Yaskawa INFORM job: A_ROOF_SIDE_0617_2_PAINT_33.JBI

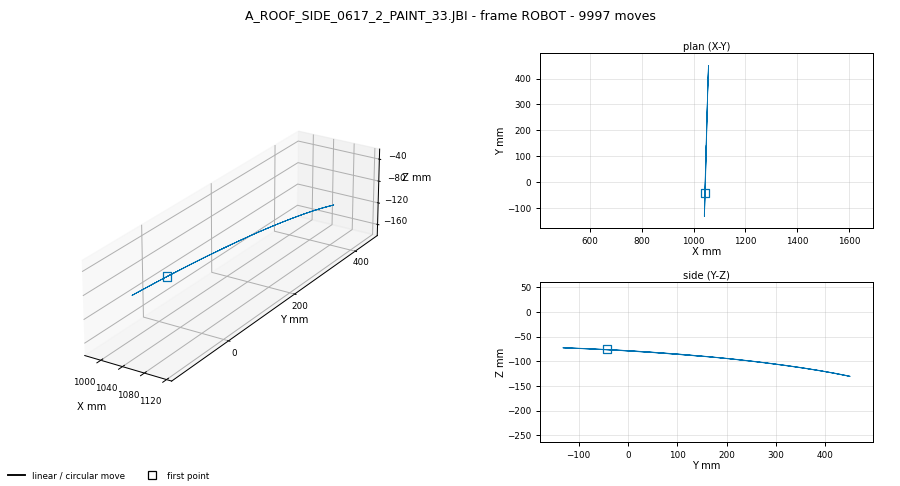
[picture p0: tool path of A_ROOF_SIDE_0617_2_PAINT_33.JBI in frame ROBOT, 9997 of 9997 moves have a stored position in this frame; points joined in program order, loops and branches not executed]
/JOB
//NAME A_ROOF_SIDE_0617_2_PAINT33
//POS
///NPOS 9997,0,0,0,0,0
///TOOL 1
///USER 0
///POSTYPE ROBOT
///RECTAN
///RCONF 1,0,0,0,0,0,0,0,0,0,0,0,0,0,0,0,0,0,0,0,0,0,0,0
C00000=1044.630,-42.557,-75.520,169.628,34.372,156.485
C00001=1044.636,-42.308,-75.534,169.630,34.372,156.485
C00002=1044.642,-42.058,-75.546,169.632,34.373,156.485
C00003=1044.648,-41.809,-75.559,169.634,34.375,156.485
C00004=1044.655,-41.560,-75.572,169.636,34.375,156.486
C00005=1044.661,-41.310,-75.585,169.638,34.376,156.486
C00006=1044.667,-41.061,-75.598,169.640,34.377,156.486
C00007=1044.674,-40.810,-75.611,169.642,34.378,156.486
C00008=1044.680,-40.561,-75.624,169.645,34.379,156.486
C00009=1044.687,-40.311,-75.636,169.647,34.380,156.486
C00010=1044.693,-40.062,-75.649,169.649,34.381,156.486
C00011=1044.699,-39.813,-75.663,169.651,34.382,156.486
C00012=1044.706,-39.562,-75.676,169.653,34.383,156.486
C00013=1044.712,-39.313,-75.689,169.656,34.384,156.487
C00014=1044.718,-39.063,-75.701,169.658,34.385,156.487
C00015=1044.725,-38.814,-75.714,169.660,34.385,156.487
C00016=1044.731,-38.565,-75.727,169.662,34.387,156.487
C00017=1044.738,-38.314,-75.740,169.664,34.388,156.487
C00018=1044.744,-38.065,-75.754,169.666,34.389,156.487
C00019=1044.749,-37.816,-75.767,169.668,34.390,156.487
C00020=1044.755,-37.566,-75.781,169.670,34.391,156.488
C00021=1044.761,-37.316,-75.793,169.672,34.392,156.488
C00022=1044.768,-37.067,-75.807,169.674,34.393,156.488
C00023=1044.774,-36.817,-75.820,169.677,34.394,156.488
C00024=1044.781,-36.568,-75.833,169.679,34.395,156.488
C00025=1044.787,-36.318,-75.846,169.681,34.396,156.488
C00026=1044.793,-36.069,-75.859,169.683,34.398,156.488
C00027=1044.800,-35.819,-75.873,169.685,34.398,156.489
C00028=1044.806,-35.538,-75.887,169.687,34.400,156.489
C00029=1044.813,-35.257,-75.903,169.689,34.401,156.489
C00030=1044.820,-34.977,-75.917,169.692,34.402,156.489
C00031=1044.828,-34.695,-75.932,169.694,34.403,156.489
C00032=1044.834,-34.446,-75.945,169.696,34.405,156.489
C00033=1044.840,-34.197,-75.958,169.698,34.405,156.489
C00034=1044.846,-33.947,-75.972,169.700,34.407,156.490
C00035=1044.852,-33.697,-75.986,169.702,34.407,156.490
C00036=1044.858,-33.448,-75.998,169.704,34.409,156.490
C00037=1044.864,-33.198,-76.012,169.706,34.410,156.490
C00038=1044.871,-32.949,-76.025,169.708,34.411,156.490
C00039=1044.878,-32.699,-76.039,169.710,34.412,156.490
C00040=1044.884,-32.450,-76.052,169.712,34.413,156.491
C00041=1044.890,-32.200,-76.065,169.714,34.414,156.491
C00042=1044.897,-31.951,-76.079,169.716,34.415,156.491
C00043=1044.903,-31.701,-76.092,169.718,34.416,156.491
C00044=1044.909,-31.452,-76.105,169.720,34.417,156.491
C00045=1044.915,-31.201,-76.119,169.722,34.418,156.491
C00046=1044.921,-30.952,-76.132,169.724,34.419,156.491
C00047=1044.927,-30.703,-76.145,169.726,34.420,156.491
C00048=1044.934,-30.453,-76.159,169.728,34.422,156.492
C00049=1044.940,-30.203,-76.172,169.730,34.422,156.492
C00050=1044.947,-29.954,-76.186,169.732,34.424,156.492
C00051=1044.953,-29.704,-76.199,169.734,34.424,156.492
C00052=1044.960,-29.455,-76.212,169.736,34.426,156.492
C00053=1044.966,-29.206,-76.226,169.739,34.427,156.492
C00054=1044.972,-28.955,-76.240,169.741,34.428,156.493
C00055=1044.978,-28.706,-76.253,169.743,34.429,156.493
C00056=1044.984,-28.457,-76.267,169.745,34.430,156.493
C00057=1044.991,-28.207,-76.280,169.748,34.431,156.493
C00058=1044.997,-27.958,-76.293,169.750,34.432,156.493
C00059=1045.004,-27.708,-76.307,169.752,34.434,156.493
C00060=1045.010,-27.458,-76.320,169.754,34.434,156.493
C00061=1045.017,-27.209,-76.334,169.756,34.436,156.494
C00062=1045.023,-26.959,-76.348,169.758,34.436,156.494
C00063=1045.029,-26.710,-76.361,169.760,34.438,156.494
C00064=1045.035,-26.461,-76.375,169.762,34.439,156.494
C00065=1045.042,-26.211,-76.389,169.763,34.440,156.494
C00066=1045.048,-25.961,-76.403,169.765,34.441,156.494
C00067=1045.054,-25.712,-76.416,169.767,34.443,156.495
C00068=1045.060,-25.462,-76.430,169.769,34.444,156.495
C00069=1045.066,-25.213,-76.443,169.771,34.445,156.495
C00070=1045.073,-24.963,-76.457,169.773,34.446,156.495
C00071=1045.079,-24.714,-76.472,169.775,34.447,156.495
C00072=1045.085,-24.464,-76.485,169.777,34.448,156.495
C00073=1045.091,-24.214,-76.499,169.779,34.450,156.496
C00074=1045.097,-23.965,-76.512,169.781,34.451,156.496
C00075=1045.104,-23.715,-76.526,169.783,34.452,156.496
C00076=1045.110,-23.465,-76.540,169.785,34.453,156.496
C00077=1045.116,-23.217,-76.554,169.787,34.454,156.496
C00078=1045.123,-22.967,-76.567,169.789,34.456,156.496
C00079=1045.128,-22.717,-76.581,169.791,34.457,156.497
C00080=1045.135,-22.467,-76.595,169.793,34.458,156.497
C00081=1045.141,-22.218,-76.610,169.795,34.459,156.497
C00082=1045.148,-21.968,-76.623,169.797,34.461,156.497
C00083=1045.154,-21.719,-76.636,169.799,34.461,156.497
C00084=1045.160,-21.469,-76.650,169.801,34.463,156.497
C00085=1045.167,-21.220,-76.665,169.804,34.464,156.498
C00086=1045.172,-20.970,-76.679,169.806,34.465,156.498
C00087=1045.179,-20.720,-76.692,169.808,34.466,156.498
C00088=1045.186,-20.472,-76.706,169.810,34.468,156.498
C00089=1045.192,-20.222,-76.720,169.812,34.469,156.498
C00090=1045.198,-19.972,-76.734,169.814,34.470,156.498
C00091=1045.204,-19.723,-76.749,169.816,34.471,156.499
C00092=1045.211,-19.441,-76.764,169.818,34.472,156.499
C00093=1045.218,-19.159,-76.780,169.820,34.474,156.499
C00094=1045.225,-18.878,-76.795,169.822,34.475,156.499
C00095=1045.232,-18.596,-76.811,169.824,34.477,156.499
C00096=1045.239,-18.347,-76.825,169.826,34.478,156.500
C00097=1045.245,-18.097,-76.839,169.828,34.479,156.500
C00098=1045.252,-17.848,-76.853,169.830,34.480,156.500
C00099=1045.258,-17.598,-76.867,169.832,34.481,156.500
C00100=1045.264,-17.348,-76.881,169.834,34.482,156.500
C00101=1045.271,-17.099,-76.895,169.836,34.484,156.500
C00102=1045.277,-16.849,-76.909,169.838,34.485,156.501
C00103=1045.284,-16.600,-76.923,169.840,34.486,156.501
C00104=1045.290,-16.350,-76.937,169.842,34.487,156.501
C00105=1045.296,-16.101,-76.951,169.844,34.488,156.501
C00106=1045.303,-15.851,-76.965,169.846,34.490,156.501
C00107=1045.308,-15.602,-76.979,169.848,34.491,156.502
C00108=1045.316,-15.352,-76.993,169.850,34.492,156.502
C00109=1045.322,-15.102,-77.007,169.852,34.493,156.502
C00110=1045.327,-14.853,-77.022,169.854,34.495,156.502
C00111=1045.334,-14.603,-77.036,169.855,34.496,156.502
C00112=1045.340,-14.354,-77.050,169.858,34.497,156.502
C00113=1045.346,-14.104,-77.064,169.860,34.499,156.503
C00114=1045.353,-13.855,-77.078,169.862,34.500,156.503
C00115=1045.359,-13.605,-77.093,169.864,34.501,156.503
C00116=1045.365,-13.356,-77.107,169.866,34.502,156.503
C00117=1045.372,-13.107,-77.122,169.868,34.503,156.503
C00118=1045.378,-12.856,-77.136,169.870,34.505,156.504
C00119=1045.383,-12.607,-77.150,169.872,34.506,156.504
C00120=1045.390,-12.357,-77.164,169.874,34.508,156.504
C00121=1045.396,-12.109,-77.179,169.876,34.509,156.504
C00122=1045.402,-11.859,-77.194,169.877,34.510,156.504
C00123=1045.409,-11.610,-77.207,169.879,34.512,156.505
C00124=1045.415,-11.360,-77.222,169.881,34.512,156.505
C00125=1045.421,-11.110,-77.236,169.883,34.514,156.505
C00126=1045.428,-10.861,-77.250,169.885,34.515,156.505
C00127=1045.434,-10.611,-77.265,169.887,34.516,156.505
C00128=1045.440,-10.361,-77.279,169.889,34.518,156.505
C00129=1045.447,-10.112,-77.293,169.891,34.519,156.506
C00130=1045.453,-9.863,-77.308,169.893,34.521,156.506
C00131=1045.459,-9.613,-77.322,169.895,34.522,156.506
C00132=1045.466,-9.364,-77.336,169.896,34.523,156.506
C00133=1045.472,-9.114,-77.351,169.898,34.525,156.507
C00134=1045.478,-8.865,-77.366,169.900,34.525,156.507
C00135=1045.484,-8.615,-77.380,169.903,34.527,156.507
C00136=1045.491,-8.366,-77.394,169.905,34.528,156.507
C00137=1045.497,-8.117,-77.409,169.907,34.529,156.507
C00138=1045.503,-7.866,-77.423,169.909,34.531,156.507
C00139=1045.510,-7.617,-77.438,169.911,34.532,156.508
C00140=1045.516,-7.368,-77.452,169.913,34.534,156.508
C00141=1045.522,-7.118,-77.467,169.914,34.535,156.508
C00142=1045.528,-6.868,-77.481,169.916,34.536,156.508
C00143=1045.535,-6.620,-77.495,169.918,34.537,156.508
C00144=1045.541,-6.370,-77.510,169.920,34.538,156.509
C00145=1045.548,-6.120,-77.525,169.922,34.540,156.509
C00146=1045.555,-5.871,-77.540,169.924,34.541,156.509
C00147=1045.560,-5.621,-77.553,169.926,34.542,156.509
C00148=1045.566,-5.372,-77.568,169.928,34.544,156.509
C00149=1045.573,-5.122,-77.583,169.929,34.545,156.510
C00150=1045.580,-4.873,-77.598,169.931,34.546,156.510
C00151=1045.586,-4.624,-77.612,169.933,34.548,156.510
C00152=1045.592,-4.373,-77.627,169.935,34.549,156.510
C00153=1045.598,-4.124,-77.641,169.937,34.551,156.510
C00154=1045.605,-3.875,-77.655,169.939,34.551,156.510
C00155=1045.611,-3.625,-77.670,169.941,34.553,156.511
C00156=1045.618,-3.342,-77.687,169.943,34.555,156.511
C00157=1045.626,-3.059,-77.704,169.946,34.556,156.511
C00158=1045.632,-2.775,-77.721,169.948,34.557,156.511
C00159=1045.639,-2.492,-77.738,169.950,34.559,156.512
C00160=1045.646,-2.243,-77.753,169.952,34.561,156.512
C00161=1045.651,-1.994,-77.767,169.954,34.562,156.512
C00162=1045.658,-1.744,-77.782,169.956,34.563,156.512
C00163=1045.664,-1.495,-77.797,169.957,34.565,156.513
C00164=1045.671,-1.245,-77.812,169.959,34.566,156.513
C00165=1045.676,-0.996,-77.827,169.961,34.567,156.513
C00166=1045.683,-0.746,-77.842,169.963,34.569,156.513
C00167=1045.689,-0.497,-77.857,169.965,34.570,156.513
C00168=1045.696,-0.247,-77.872,169.967,34.572,156.514
C00169=1045.701,0.002,-77.886,169.968,34.573,156.514
C00170=1045.708,0.252,-77.901,169.970,34.575,156.514
C00171=1045.713,0.502,-77.917,169.972,34.576,156.514
C00172=1045.720,0.751,-77.932,169.974,34.578,156.515
C00173=1045.726,1.000,-77.946,169.976,34.579,156.515
C00174=1045.732,1.250,-77.961,169.978,34.580,156.515
C00175=1045.738,1.500,-77.976,169.979,34.582,156.515
C00176=1045.745,1.749,-77.991,169.982,34.583,156.515
C00177=1045.750,1.998,-78.006,169.984,34.584,156.516
C00178=1045.757,2.248,-78.021,169.986,34.586,156.516
C00179=1045.763,2.497,-78.035,169.988,34.588,156.516
C00180=1045.770,2.746,-78.051,169.989,34.589,156.516
C00181=1045.776,2.996,-78.066,169.991,34.590,156.517
C00182=1045.783,3.246,-78.081,169.993,34.592,156.517
C00183=1045.788,3.495,-78.096,169.995,34.593,156.517
C00184=1045.795,3.744,-78.111,169.997,34.594,156.517
C00185=1045.801,3.994,-78.126,169.999,34.596,156.517
C00186=1045.807,4.244,-78.141,170.000,34.597,156.518
C00187=1045.814,4.493,-78.157,170.002,34.598,156.518
C00188=1045.820,4.743,-78.172,170.004,34.600,156.518
C00189=1045.826,4.992,-78.186,170.006,34.601,156.518
C00190=1045.832,5.241,-78.201,170.008,34.603,156.518
C00191=1045.839,5.491,-78.216,170.009,34.604,156.519
C00192=1045.845,5.740,-78.232,170.011,34.606,156.519
C00193=1045.852,5.990,-78.247,170.013,34.607,156.519
C00194=1045.858,6.239,-78.262,170.016,34.608,156.519
C00195=1045.864,6.489,-78.277,170.018,34.610,156.520
C00196=1045.869,6.738,-78.292,170.020,34.611,156.520
C00197=1045.876,6.987,-78.307,170.021,34.612,156.520
C00198=1045.882,7.237,-78.322,170.023,34.614,156.520
C00199=1045.889,7.487,-78.337,170.025,34.615,156.520
C00200=1045.895,7.736,-78.352,170.027,34.617,156.521
C00201=1045.902,7.985,-78.368,170.029,34.618,156.521
C00202=1045.908,8.235,-78.383,170.030,34.620,156.521
C00203=1045.915,8.485,-78.398,170.032,34.621,156.521
C00204=1045.921,8.734,-78.414,170.034,34.623,156.522
C00205=1045.927,8.984,-78.429,170.036,34.624,156.522
C00206=1045.933,9.233,-78.444,170.038,34.625,156.522
C00207=1045.940,9.482,-78.460,170.039,34.627,156.522
C00208=1045.946,9.731,-78.474,170.041,34.628,156.522
C00209=1045.952,9.981,-78.489,170.043,34.629,156.523
C00210=1045.959,10.230,-78.505,170.045,34.631,156.523
C00211=1045.965,10.480,-78.520,170.047,34.633,156.523
C00212=1045.971,10.730,-78.535,170.049,34.634,156.523
C00213=1045.978,10.979,-78.551,170.051,34.635,156.524
C00214=1045.984,11.228,-78.566,170.053,34.637,156.524
C00215=1045.990,11.478,-78.581,170.055,34.638,156.524
C00216=1045.997,11.727,-78.597,170.057,34.639,156.524
C00217=1046.004,11.977,-78.612,170.058,34.641,156.524
C00218=1046.010,12.226,-78.627,170.060,34.642,156.525
C00219=1046.016,12.476,-78.643,170.062,34.643,156.525
C00220=1046.023,12.761,-78.660,170.064,34.645,156.525
C00221=1046.031,13.046,-78.678,170.066,34.647,156.525
C00222=1046.038,13.331,-78.695,170.068,34.648,156.526
C00223=1046.045,13.616,-78.713,170.070,34.650,156.526
C00224=1046.052,13.865,-78.728,170.072,34.651,156.526
C00225=1046.058,14.115,-78.743,170.074,34.653,156.526
C00226=1046.065,14.364,-78.759,170.076,34.654,156.526
C00227=1046.070,14.614,-78.774,170.077,34.655,156.527
C00228=1046.077,14.863,-78.790,170.080,34.657,156.527
C00229=1046.083,15.113,-78.806,170.082,34.659,156.527
C00230=1046.090,15.362,-78.821,170.084,34.660,156.527
C00231=1046.096,15.611,-78.837,170.085,34.661,156.528
C00232=1046.102,15.861,-78.852,170.087,34.663,156.528
C00233=1046.109,16.110,-78.868,170.089,34.665,156.528
C00234=1046.114,16.360,-78.883,170.091,34.666,156.528
C00235=1046.121,16.609,-78.899,170.092,34.667,156.529
C00236=1046.127,16.859,-78.914,170.094,34.669,156.529
C00237=1046.133,17.108,-78.930,170.096,34.671,156.529
C00238=1046.140,17.357,-78.946,170.098,34.672,156.529
C00239=1046.146,17.607,-78.962,170.099,34.673,156.530
C00240=1046.152,17.856,-78.977,170.101,34.675,156.530
C00241=1046.159,18.107,-78.992,170.103,34.677,156.530
C00242=1046.165,18.356,-79.009,170.105,34.678,156.530
C00243=1046.172,18.605,-79.024,170.106,34.679,156.530
C00244=1046.177,18.855,-79.040,170.109,34.681,156.531
C00245=1046.184,19.104,-79.056,170.111,34.682,156.531
C00246=1046.191,19.353,-79.071,170.113,34.684,156.531
C00247=1046.197,19.603,-79.087,170.114,34.685,156.531
C00248=1046.203,19.852,-79.102,170.116,34.687,156.532
C00249=1046.209,20.101,-79.119,170.118,34.688,156.532
C00250=1046.216,20.351,-79.134,170.120,34.690,156.532
C00251=1046.221,20.600,-79.150,170.121,34.691,156.532
C00252=1046.228,20.849,-79.166,170.123,34.693,156.533
C00253=1046.234,21.099,-79.182,170.125,34.695,156.533
C00254=1046.240,21.349,-79.197,170.127,34.696,156.533
C00255=1046.246,21.598,-79.213,170.128,34.697,156.533
C00256=1046.253,21.848,-79.230,170.130,34.699,156.534
C00257=1046.260,22.097,-79.245,170.132,34.700,156.534
C00258=1046.265,22.347,-79.261,170.134,34.702,156.534
C00259=1046.272,22.596,-79.277,170.135,34.703,156.534
C00260=1046.278,22.845,-79.293,170.138,34.705,156.535
C00261=1046.285,23.094,-79.308,170.140,34.706,156.535
C00262=1046.291,23.344,-79.325,170.142,34.708,156.535
C00263=1046.296,23.594,-79.340,170.143,34.709,156.535
C00264=1046.303,23.843,-79.356,170.145,34.711,156.536
C00265=1046.310,24.093,-79.373,170.147,34.712,156.536
C00266=1046.316,24.342,-79.388,170.148,34.714,156.536
C00267=1046.322,24.591,-79.404,170.150,34.716,156.536
C00268=1046.329,24.841,-79.419,170.152,34.717,156.537
C00269=1046.334,25.090,-79.436,170.154,34.718,156.537
C00270=1046.340,25.339,-79.452,170.155,34.720,156.537
C00271=1046.347,25.588,-79.468,170.157,34.722,156.537
C00272=1046.354,25.839,-79.484,170.159,34.723,156.538
C00273=1046.360,26.088,-79.500,170.161,34.724,156.538
C00274=1046.366,26.337,-79.516,170.163,34.726,156.538
C00275=1046.373,26.586,-79.532,170.165,34.728,156.538
C00276=1046.379,26.835,-79.548,170.167,34.729,156.538
C00277=1046.385,27.085,-79.564,170.168,34.730,156.539
C00278=1046.392,27.335,-79.580,170.170,34.732,156.539
C00279=1046.398,27.584,-79.596,170.172,34.734,156.539
C00280=1046.404,27.834,-79.612,170.174,34.735,156.539
C00281=1046.410,28.083,-79.628,170.175,34.737,156.540
C00282=1046.416,28.332,-79.644,170.177,34.738,156.540
C00283=1046.423,28.582,-79.661,170.179,34.740,156.540
C00284=1046.430,28.868,-79.679,170.181,34.741,156.541
C00285=1046.438,29.155,-79.698,170.183,34.743,156.541
C00286=1046.445,29.440,-79.716,170.185,34.745,156.541
C00287=1046.451,29.727,-79.735,170.187,34.747,156.541
C00288=1046.458,29.977,-79.751,170.189,34.749,156.542
C00289=1046.464,30.226,-79.767,170.191,34.750,156.542
C00290=1046.470,30.476,-79.783,170.193,34.751,156.542
C00291=1046.476,30.725,-79.800,170.194,34.753,156.542
C00292=1046.482,30.974,-79.817,170.196,34.755,156.543
C00293=1046.490,31.224,-79.833,170.198,34.756,156.543
C00294=1046.496,31.473,-79.849,170.200,34.758,156.543
C00295=1046.502,31.722,-79.865,170.201,34.759,156.543
C00296=1046.507,31.972,-79.881,170.203,34.761,156.544
C00297=1046.514,32.222,-79.898,170.205,34.763,156.544
C00298=1046.521,32.471,-79.914,170.206,34.764,156.544
C00299=1046.527,32.720,-79.930,170.208,34.766,156.545
C00300=1046.533,32.969,-79.946,170.210,34.767,156.545
C00301=1046.539,33.219,-79.963,170.212,34.768,156.545
C00302=1046.545,33.468,-79.980,170.214,34.770,156.545
C00303=1046.552,33.717,-79.995,170.216,34.772,156.545
C00304=1046.558,33.967,-80.012,170.218,34.774,156.546
C00305=1046.565,34.217,-80.028,170.219,34.775,156.546
C00306=1046.571,34.466,-80.044,170.221,34.776,156.546
C00307=1046.577,34.715,-80.061,170.223,34.778,156.547
C00308=1046.583,34.964,-80.078,170.224,34.780,156.547
C00309=1046.590,35.214,-80.094,170.226,34.781,156.547
C00310=1046.596,35.463,-80.110,170.228,34.783,156.547
C00311=1046.602,35.713,-80.126,170.229,34.784,156.548
C00312=1046.609,35.963,-80.143,170.231,34.786,156.548
C00313=1046.615,36.211,-80.160,170.233,34.788,156.548
C00314=1046.621,36.461,-80.176,170.236,34.789,156.548
C00315=1046.628,36.710,-80.192,170.237,34.791,156.549
C00316=1046.634,36.960,-80.208,170.239,34.792,156.549
C00317=1046.640,37.208,-80.225,170.241,34.793,156.549
C00318=1046.646,37.458,-80.242,170.242,34.795,156.549
C00319=1046.653,37.708,-80.258,170.244,34.797,156.550
C00320=1046.659,37.957,-80.275,170.246,34.799,156.550
C00321=1046.665,38.206,-80.291,170.247,34.800,156.550
C00322=1046.671,38.456,-80.308,170.249,34.801,156.550
C00323=1046.677,38.705,-80.324,170.251,34.803,156.551
C00324=1046.684,38.954,-80.341,170.252,34.805,156.551
C00325=1046.690,39.204,-80.358,170.254,34.807,156.551
C00326=1046.697,39.453,-80.375,170.256,34.808,156.551
C00327=1046.702,39.702,-80.391,170.258,34.810,156.552
C00328=1046.709,39.952,-80.408,170.260,34.811,156.552
C00329=1046.715,40.201,-80.425,170.262,34.813,156.552
C00330=1046.720,40.451,-80.442,170.263,34.814,156.553
C00331=1046.727,40.701,-80.458,170.265,34.816,156.553
C00332=1046.733,40.949,-80.475,170.267,34.818,156.553
C00333=1046.739,41.199,-80.491,170.268,34.820,156.553
C00334=1046.746,41.448,-80.509,170.270,34.821,156.554
C00335=1046.752,41.698,-80.525,170.272,34.822,156.554
C00336=1046.758,41.947,-80.541,170.273,34.824,156.554
C00337=1046.765,42.196,-80.559,170.275,34.825,156.554
C00338=1046.771,42.446,-80.575,170.277,34.827,156.555
C00339=1046.777,42.694,-80.592,170.279,34.829,156.555
C00340=1046.784,42.944,-80.609,170.281,34.831,156.555
C00341=1046.790,43.193,-80.625,170.283,34.832,156.555
C00342=1046.796,43.443,-80.642,170.285,34.834,156.556
C00343=1046.802,43.692,-80.660,170.286,34.835,156.556
C00344=1046.808,43.942,-80.676,170.288,34.837,156.556
C00345=1046.815,44.191,-80.693,170.289,34.839,156.557
C00346=1046.820,44.441,-80.710,170.291,34.840,156.557
C00347=1046.826,44.689,-80.727,170.293,34.842,156.557
C00348=1046.833,44.977,-80.747,170.295,34.844,156.558
C00349=1046.840,45.263,-80.767,170.297,34.846,156.558
C00350=1046.848,45.549,-80.785,170.298,34.848,156.558
C00351=1046.855,45.835,-80.805,170.301,34.850,156.558
C00352=1046.861,46.085,-80.822,170.303,34.852,156.559
C00353=1046.867,46.334,-80.839,170.305,34.854,156.559
C00354=1046.873,46.583,-80.856,170.306,34.855,156.559
C00355=1046.879,46.833,-80.874,170.308,34.857,156.560
C00356=1046.885,47.082,-80.891,170.310,34.858,156.560
C00357=1046.891,47.331,-80.907,170.311,34.860,156.560
C00358=1046.897,47.581,-80.925,170.313,34.861,156.560
C00359=1046.904,47.830,-80.942,170.314,34.863,156.561
C00360=1046.910,48.080,-80.958,170.316,34.865,156.561
C00361=1046.916,48.329,-80.976,170.318,34.867,156.561
C00362=1046.922,48.578,-80.993,170.320,34.868,156.562
C00363=1046.928,48.827,-81.010,170.322,34.870,156.562
C00364=1046.934,49.076,-81.027,170.324,34.872,156.562
C00365=1046.941,49.326,-81.044,170.325,34.873,156.562
C00366=1046.947,49.575,-81.061,170.327,34.875,156.563
C00367=1046.953,49.825,-81.079,170.329,34.876,156.563
C00368=1046.959,50.074,-81.096,170.330,34.878,156.563
C00369=1046.966,50.324,-81.112,170.332,34.880,156.564
C00370=1046.971,50.573,-81.130,170.334,34.882,156.564
C00371=1046.978,50.822,-81.147,170.335,34.883,156.564
C00372=1046.984,51.071,-81.164,170.337,34.885,156.564
C00373=1046.990,51.321,-81.181,170.340,34.887,156.565
C00374=1046.996,51.570,-81.198,170.341,34.888,156.565
C00375=1047.003,51.819,-81.216,170.343,34.890,156.565
C00376=1047.009,52.068,-81.233,170.344,34.891,156.565
C00377=1047.015,52.318,-81.249,170.346,34.893,156.566
C00378=1047.021,52.568,-81.267,170.348,34.895,156.566
C00379=1047.028,52.817,-81.285,170.349,34.896,156.566
C00380=1047.034,53.066,-81.302,170.351,34.898,156.567
C00381=1047.040,53.315,-81.320,170.353,34.900,156.567
C00382=1047.046,53.565,-81.336,170.354,34.902,156.567
C00383=1047.053,53.814,-81.353,170.356,34.903,156.567
C00384=1047.058,54.063,-81.371,170.359,34.905,156.568
C00385=1047.065,54.313,-81.388,170.360,34.906,156.568
C00386=1047.071,54.562,-81.406,170.362,34.908,156.568
C00387=1047.078,54.811,-81.423,170.364,34.909,156.568
C00388=1047.084,55.060,-81.440,170.365,34.911,156.569
C00389=1047.090,55.310,-81.457,170.367,34.913,156.569
C00390=1047.096,55.559,-81.474,170.369,34.915,156.569
C00391=1047.103,55.808,-81.492,170.370,34.916,156.570
C00392=1047.109,56.058,-81.509,170.372,34.918,156.570
C00393=1047.115,56.307,-81.526,170.374,34.919,156.570
C00394=1047.121,56.557,-81.544,170.375,34.921,156.570
C00395=1047.128,56.805,-81.561,170.377,34.922,156.571
C00396=1047.134,57.055,-81.579,170.379,34.924,156.571
C00397=1047.140,57.304,-81.596,170.381,34.926,156.571
C00398=1047.147,57.553,-81.614,170.383,34.928,156.572
C00399=1047.153,57.804,-81.631,170.384,34.929,156.572
C00400=1047.159,58.052,-81.648,170.386,34.931,156.572
C00401=1047.166,58.302,-81.665,170.388,34.932,156.572
C00402=1047.171,58.551,-81.683,170.389,34.934,156.573
C00403=1047.178,58.800,-81.700,170.391,34.935,156.573
C00404=1047.184,59.050,-81.718,170.393,34.937,156.573
C00405=1047.190,59.299,-81.735,170.394,34.939,156.573
C00406=1047.197,59.548,-81.753,170.397,34.941,156.574
C00407=1047.203,59.798,-81.770,170.399,34.942,156.574
C00408=1047.210,60.047,-81.787,170.400,34.944,156.574
C00409=1047.216,60.296,-81.805,170.402,34.945,156.575
C00410=1047.223,60.546,-81.822,170.404,34.947,156.575
C00411=1047.228,60.795,-81.840,170.405,34.948,156.575
C00412=1047.236,61.081,-81.860,170.407,34.950,156.575
C00413=1047.244,61.366,-81.880,170.409,34.952,156.576
C00414=1047.251,61.652,-81.900,170.411,34.954,156.576
C00415=1047.258,61.939,-81.921,170.413,34.956,156.576
C00416=1047.264,62.188,-81.938,170.415,34.958,156.577
C00417=1047.271,62.438,-81.956,170.417,34.959,156.577
C00418=1047.278,62.687,-81.973,170.419,34.961,156.577
C00419=1047.283,62.936,-81.990,170.420,34.963,156.578
C00420=1047.290,63.185,-82.008,170.422,34.964,156.578
C00421=1047.296,63.435,-82.026,170.424,34.966,156.578
C00422=1047.303,63.684,-82.044,170.425,34.967,156.578
C00423=1047.309,63.933,-82.061,170.427,34.969,156.579
C00424=1047.316,64.182,-82.079,170.429,34.970,156.579
C00425=1047.322,64.432,-82.097,170.430,34.972,156.579
C00426=1047.327,64.681,-82.114,170.432,34.974,156.579
C00427=1047.334,64.931,-82.132,170.434,34.976,156.580
C00428=1047.341,65.180,-82.150,170.436,34.978,156.580
C00429=1047.346,65.429,-82.168,170.438,34.979,156.580
C00430=1047.352,65.679,-82.186,170.440,34.981,156.581
C00431=1047.359,65.928,-82.203,170.441,34.982,156.581
C00432=1047.365,66.177,-82.221,170.443,34.984,156.581
C00433=1047.371,66.426,-82.239,170.444,34.986,156.581
C00434=1047.378,66.676,-82.257,170.446,34.987,156.582
C00435=1047.384,66.925,-82.275,170.448,34.989,156.582
C00436=1047.389,67.174,-82.292,170.449,34.990,156.582
C00437=1047.396,67.423,-82.311,170.451,34.992,156.583
C00438=1047.403,67.673,-82.328,170.454,34.994,156.583
C00439=1047.408,67.922,-82.346,170.455,34.996,156.583
C00440=1047.415,68.171,-82.364,170.457,34.998,156.583
C00441=1047.421,68.421,-82.382,170.458,34.999,156.584
C00442=1047.428,68.670,-82.400,170.460,35.001,156.584
C00443=1047.433,68.919,-82.418,170.462,35.003,156.584
C00444=1047.440,69.168,-82.436,170.463,35.004,156.585
C00445=1047.446,69.418,-82.454,170.465,35.006,156.585
C00446=1047.453,69.667,-82.472,170.467,35.008,156.585
C00447=1047.458,69.916,-82.489,170.468,35.009,156.585
C00448=1047.465,70.166,-82.507,170.471,35.011,156.586
C00449=1047.471,70.415,-82.526,170.473,35.013,156.586
C00450=1047.476,70.664,-82.543,170.474,35.014,156.586
C00451=1047.483,70.913,-82.562,170.476,35.016,156.587
C00452=1047.489,71.163,-82.580,170.477,35.018,156.587
C00453=1047.495,71.413,-82.598,170.479,35.019,156.587
C00454=1047.502,71.661,-82.616,170.481,35.021,156.588
C00455=1047.508,71.910,-82.634,170.482,35.023,156.588
C00456=1047.514,72.159,-82.652,170.484,35.025,156.588
C00457=1047.520,72.409,-82.670,170.486,35.027,156.588
C00458=1047.526,72.658,-82.688,170.488,35.028,156.589
C00459=1047.532,72.907,-82.706,170.490,35.030,156.589
C00460=1047.539,73.157,-82.725,170.491,35.032,156.589
C00461=1047.545,73.406,-82.743,170.493,35.034,156.590
C00462=1047.551,73.655,-82.762,170.495,35.035,156.590
C00463=1047.557,73.904,-82.779,170.496,35.037,156.590
C00464=1047.563,74.154,-82.798,170.498,35.039,156.591
C00465=1047.569,74.403,-82.816,170.500,35.040,156.591
C00466=1047.576,74.652,-82.834,170.501,35.042,156.591
C00467=1047.583,74.902,-82.852,170.504,35.044,156.591
C00468=1047.588,75.150,-82.870,170.505,35.045,156.592
C00469=1047.595,75.400,-82.888,170.507,35.047,156.592
C00470=1047.601,75.649,-82.907,170.509,35.049,156.592
C00471=1047.607,75.899,-82.925,170.510,35.050,156.593
C00472=1047.614,76.148,-82.943,170.512,35.052,156.593
C00473=1047.620,76.398,-82.961,170.514,35.054,156.593
C00474=1047.626,76.646,-82.979,170.515,35.056,156.594
C00475=1047.632,76.895,-82.998,170.517,35.057,156.594
C00476=1047.639,77.182,-83.018,170.519,35.059,156.594
C00477=1047.646,77.468,-83.040,170.522,35.061,156.595
C00478=1047.653,77.753,-83.061,170.523,35.063,156.595
C00479=1047.660,78.039,-83.082,170.525,35.065,156.595
C00480=1047.667,78.288,-83.101,170.527,35.067,156.596
C00481=1047.673,78.538,-83.119,170.529,35.068,156.596
C00482=1047.679,78.786,-83.137,170.530,35.070,156.596
C00483=1047.684,79.036,-83.156,170.532,35.072,156.596
C00484=1047.691,79.286,-83.174,170.533,35.074,156.597
C00485=1047.697,79.535,-83.193,170.535,35.075,156.597
C00486=1047.703,79.784,-83.211,170.538,35.077,156.597
C00487=1047.710,80.033,-83.230,170.539,35.079,156.598
C00488=1047.715,80.282,-83.248,170.541,35.081,156.598
C00489=1047.721,80.531,-83.267,170.543,35.083,156.598
C00490=1047.728,80.781,-83.285,170.544,35.084,156.599
C00491=1047.734,81.030,-83.304,170.546,35.086,156.599
C00492=1047.740,81.279,-83.322,170.547,35.088,156.599
C00493=1047.746,81.529,-83.341,170.549,35.090,156.599
C00494=1047.752,81.778,-83.360,170.551,35.092,156.600
C00495=1047.759,82.027,-83.379,170.553,35.093,156.600
C00496=1047.764,82.276,-83.396,170.555,35.095,156.600
C00497=1047.771,82.525,-83.415,170.556,35.097,156.601
C00498=1047.777,82.774,-83.433,170.558,35.099,156.601
C00499=1047.783,83.024,-83.453,170.560,35.100,156.601
C00500=1047.789,83.273,-83.471,170.561,35.102,156.602
C00501=1047.796,83.522,-83.490,170.563,35.104,156.602
C00502=1047.802,83.772,-83.508,170.565,35.106,156.602
C00503=1047.807,84.021,-83.527,170.566,35.107,156.603
C00504=1047.814,84.270,-83.546,170.569,35.109,156.603
C00505=1047.820,84.519,-83.564,170.571,35.111,156.603
C00506=1047.826,84.768,-83.583,170.572,35.113,156.603
C00507=1047.832,85.017,-83.601,170.574,35.115,156.604
C00508=1047.838,85.266,-83.621,170.575,35.116,156.604
C00509=1047.845,85.516,-83.639,170.577,35.118,156.604
C00510=1047.851,85.765,-83.657,170.579,35.120,156.605
C00511=1047.857,86.014,-83.676,170.580,35.122,156.605
C00512=1047.863,86.264,-83.695,170.582,35.123,156.605
C00513=1047.869,86.513,-83.714,170.585,35.125,156.606
C00514=1047.876,86.762,-83.732,170.586,35.127,156.606
C00515=1047.882,87.011,-83.751,170.588,35.128,156.606
C00516=1047.888,87.261,-83.770,170.589,35.130,156.607
C00517=1047.894,87.510,-83.789,170.591,35.132,156.607
C00518=1047.901,87.759,-83.808,170.593,35.133,156.607
C00519=1047.907,88.008,-83.826,170.594,35.135,156.607
C00520=1047.913,88.257,-83.845,170.596,35.137,156.608
C00521=1047.919,88.507,-83.864,170.598,35.139,156.608
C00522=1047.926,88.756,-83.883,170.600,35.140,156.608
C00523=1047.932,89.005,-83.901,170.602,35.142,156.609
C00524=1047.938,89.254,-83.921,170.604,35.144,156.609
C00525=1047.944,89.503,-83.939,170.605,35.145,156.609
C00526=1047.951,89.753,-83.958,170.607,35.147,156.610
C00527=1047.957,90.002,-83.977,170.609,35.149,156.610
C00528=1047.963,90.251,-83.996,170.610,35.150,156.610
C00529=1047.969,90.500,-84.014,170.612,35.152,156.610
C00530=1047.975,90.750,-84.034,170.613,35.154,156.611
C00531=1047.981,90.999,-84.052,170.616,35.156,156.611
C00532=1047.987,91.248,-84.072,170.618,35.158,156.611
C00533=1047.993,91.497,-84.090,170.619,35.159,156.612
C00534=1047.999,91.747,-84.109,170.621,35.161,156.612
C00535=1048.006,91.995,-84.129,170.623,35.163,156.612
C00536=1048.011,92.245,-84.148,170.624,35.165,156.613
C00537=1048.018,92.494,-84.167,170.626,35.167,156.613
C00538=1048.024,92.743,-84.186,170.627,35.168,156.613
C00539=1048.030,92.992,-84.205,170.630,35.170,156.614
C00540=1048.037,93.278,-84.227,170.632,35.172,156.614
C00541=1048.045,93.564,-84.249,170.634,35.175,156.614
C00542=1048.051,93.849,-84.271,170.636,35.177,156.615
C00543=1048.058,94.136,-84.293,170.638,35.179,156.615
C00544=1048.064,94.385,-84.311,170.639,35.180,156.615
C00545=1048.070,94.634,-84.331,170.641,35.182,156.616
C00546=1048.077,94.883,-84.350,170.643,35.184,156.616
C00547=1048.082,95.133,-84.369,170.645,35.186,156.616
C00548=1048.089,95.382,-84.388,170.647,35.187,156.617
C00549=1048.095,95.630,-84.408,170.648,35.189,156.617
C00550=1048.101,95.880,-84.427,170.650,35.191,156.617
C00551=1048.107,96.129,-84.446,170.652,35.193,156.618
C00552=1048.114,96.379,-84.465,170.653,35.194,156.618
C00553=1048.120,96.628,-84.485,170.655,35.196,156.618
C00554=1048.126,96.877,-84.503,170.657,35.198,156.619
C00555=1048.132,97.126,-84.523,170.658,35.200,156.619
C00556=1048.138,97.376,-84.542,170.661,35.201,156.619
C00557=1048.144,97.624,-84.561,170.663,35.203,156.619
C00558=1048.150,97.874,-84.581,170.664,35.205,156.620
C00559=1048.156,98.123,-84.599,170.666,35.207,156.620
C00560=1048.162,98.371,-84.619,170.668,35.209,156.620
C00561=1048.170,98.621,-84.638,170.669,35.210,156.621
C00562=1048.175,98.871,-84.657,170.671,35.212,156.621
C00563=1048.182,99.119,-84.677,170.673,35.214,156.621
C00564=1048.188,99.369,-84.696,170.675,35.216,156.622
C00565=1048.194,99.617,-84.716,170.677,35.217,156.622
C00566=1048.200,99.867,-84.735,170.678,35.219,156.622
C00567=1048.206,100.116,-84.754,170.680,35.221,156.623
C00568=1048.213,100.365,-84.774,170.682,35.223,156.623
C00569=1048.219,100.615,-84.793,170.683,35.224,156.623
C00570=1048.224,100.864,-84.812,170.685,35.226,156.624
C00571=1048.230,101.113,-84.832,170.687,35.228,156.624
C00572=1048.237,101.362,-84.851,170.689,35.230,156.624
C00573=1048.243,101.611,-84.871,170.691,35.232,156.625
C00574=1048.249,101.860,-84.890,170.693,35.234,156.625
C00575=1048.255,102.110,-84.910,170.694,35.235,156.625
C00576=1048.261,102.359,-84.929,170.696,35.237,156.625
C00577=1048.268,102.608,-84.949,170.698,35.239,156.626
C00578=1048.273,102.857,-84.968,170.699,35.241,156.626
C00579=1048.279,103.106,-84.988,170.701,35.243,156.626
C00580=1048.285,103.355,-85.007,170.704,35.245,156.627
C00581=1048.291,103.604,-85.027,170.705,35.247,156.627
C00582=1048.298,103.854,-85.046,170.707,35.249,156.628
C00583=1048.304,104.103,-85.066,170.708,35.250,156.628
C00584=1048.310,104.352,-85.086,170.710,35.252,156.628
C00585=1048.316,104.601,-85.105,170.712,35.254,156.628
C00586=1048.322,104.850,-85.125,170.713,35.256,156.629
C00587=1048.327,105.099,-85.145,170.715,35.257,156.629
C00588=1048.335,105.349,-85.164,170.718,35.259,156.629
C00589=1048.340,105.598,-85.184,170.719,35.261,156.630
C00590=1048.346,105.847,-85.204,170.721,35.263,156.630
C00591=1048.352,106.096,-85.223,170.723,35.265,156.630
C00592=1048.358,106.345,-85.243,170.724,35.266,156.631
C00593=1048.365,106.595,-85.263,170.726,35.268,156.631
C00594=1048.371,106.843,-85.282,170.728,35.270,156.631
C00595=1048.377,107.093,-85.302,170.729,35.272,156.632
C00596=1048.383,107.341,-85.322,170.732,35.273,156.632
C00597=1048.390,107.591,-85.342,170.734,35.275,156.632
C00598=1048.395,107.840,-85.361,170.735,35.277,156.633
C00599=1048.401,108.089,-85.381,170.737,35.279,156.633
C00600=1048.407,108.338,-85.401,170.739,35.281,156.633
C00601=1048.414,108.588,-85.420,170.740,35.283,156.634
C00602=1048.420,108.837,-85.440,170.742,35.284,156.634
C00603=1048.426,109.085,-85.460,170.744,35.286,156.634
C00604=1048.433,109.371,-85.483,170.747,35.289,156.635
C00605=1048.440,109.657,-85.505,170.749,35.291,156.635
C00606=1048.447,109.943,-85.528,170.751,35.292,156.635
C00607=1048.455,110.229,-85.551,170.752,35.294,156.636
C00608=1048.461,110.478,-85.571,170.754,35.296,156.636
C00609=1048.467,110.728,-85.590,170.756,35.298,156.636
C00610=1048.473,110.977,-85.610,170.758,35.300,156.637
C00611=1048.479,111.225,-85.630,170.760,35.302,156.637
C00612=1048.485,111.475,-85.650,170.762,35.304,156.637
C00613=1048.491,111.724,-85.670,170.764,35.305,156.638
C00614=1048.497,111.973,-85.690,170.765,35.307,156.638
C00615=1048.503,112.222,-85.710,170.767,35.309,156.638
C00616=1048.510,112.471,-85.730,170.769,35.311,156.639
C00617=1048.516,112.720,-85.750,170.770,35.313,156.639
C00618=1048.522,112.969,-85.770,170.772,35.315,156.639
C00619=1048.528,113.219,-85.790,170.775,35.317,156.640
C00620=1048.534,113.467,-85.810,170.776,35.318,156.640
C00621=1048.540,113.717,-85.829,170.778,35.320,156.640
C00622=1048.547,113.966,-85.850,170.780,35.322,156.641
C00623=1048.553,114.215,-85.870,170.781,35.324,156.641
C00624=1048.558,114.464,-85.890,170.783,35.326,156.641
C00625=1048.564,114.713,-85.910,170.785,35.328,156.642
C00626=1048.570,114.963,-85.930,170.787,35.330,156.642
C00627=1048.576,115.212,-85.951,170.789,35.332,156.642
C00628=1048.582,115.461,-85.971,170.791,35.334,156.643
C00629=1048.588,115.710,-85.991,170.792,35.336,156.643
C00630=1048.594,115.959,-86.011,170.794,35.337,156.643
C00631=1048.599,116.208,-86.032,170.796,35.339,156.644
C00632=1048.605,116.457,-86.052,170.797,35.341,156.644
C00633=1048.612,116.706,-86.072,170.800,35.343,156.645
C00634=1048.618,116.955,-86.092,170.802,35.345,156.645
C00635=1048.623,117.204,-86.113,170.803,35.347,156.645
C00636=1048.630,117.454,-86.133,170.805,35.349,156.646
C00637=1048.636,117.703,-86.153,170.807,35.351,156.646
C00638=1048.641,117.952,-86.173,170.808,35.353,156.646
C00639=1048.648,118.201,-86.194,170.810,35.354,156.647
C00640=1048.654,118.450,-86.214,170.813,35.356,156.647
C00641=1048.660,118.698,-86.234,170.814,35.358,156.647
C00642=1048.666,118.948,-86.255,170.816,35.360,156.648
C00643=1048.672,119.197,-86.275,170.818,35.362,156.648
C00644=1048.679,119.446,-86.296,170.820,35.363,156.648
C00645=1048.684,119.696,-86.316,170.821,35.365,156.649
C00646=1048.690,119.944,-86.336,170.823,35.367,156.649
C00647=1048.696,120.194,-86.356,170.825,35.369,156.649
C00648=1048.702,120.443,-86.376,170.827,35.371,156.650
C00649=1048.708,120.692,-86.397,170.829,35.373,156.650
C00650=1048.715,120.941,-86.418,170.831,35.375,156.650
C00651=1048.721,121.189,-86.438,170.832,35.377,156.651
C00652=1048.726,121.439,-86.459,170.834,35.378,156.651
C00653=1048.732,121.688,-86.479,170.836,35.380,156.651
C00654=1048.738,121.937,-86.499,170.838,35.382,156.652
C00655=1048.745,122.186,-86.520,170.840,35.384,156.652
C00656=1048.751,122.435,-86.540,170.842,35.386,156.652
C00657=1048.757,122.684,-86.561,170.844,35.388,156.653
C00658=1048.762,122.934,-86.581,170.845,35.390,156.653
C00659=1048.769,123.183,-86.602,170.847,35.392,156.653
C00660=1048.775,123.431,-86.622,170.849,35.394,156.654
C00661=1048.781,123.681,-86.643,170.851,35.396,156.654
C00662=1048.787,123.930,-86.663,170.853,35.397,156.654
C00663=1048.793,124.179,-86.683,170.855,35.399,156.655
C00664=1048.799,124.428,-86.705,170.857,35.401,156.655
C00665=1048.805,124.677,-86.725,170.858,35.403,156.655
C00666=1048.812,124.926,-86.745,170.860,35.405,156.656
C00667=1048.817,125.175,-86.766,170.862,35.407,156.656
C00668=1048.825,125.462,-86.790,170.864,35.409,156.656
C00669=1048.832,125.747,-86.813,170.867,35.411,156.657
C00670=1048.839,126.032,-86.837,170.869,35.413,156.657
C00671=1048.846,126.318,-86.861,170.871,35.415,156.658
C00672=1048.852,126.567,-86.881,170.873,35.417,156.658
C00673=1048.858,126.816,-86.901,170.874,35.419,156.658
C00674=1048.864,127.065,-86.922,170.876,35.421,156.659
C00675=1048.870,127.314,-86.942,170.879,35.423,156.659
C00676=1048.876,127.564,-86.963,170.881,35.425,156.659
C00677=1048.883,127.812,-86.984,170.882,35.426,156.660
C00678=1048.889,128.062,-87.004,170.884,35.428,156.660
C00679=1048.895,128.310,-87.026,170.886,35.430,156.660
C00680=1048.901,128.560,-87.046,170.888,35.432,156.661
C00681=1048.908,128.809,-87.066,170.889,35.434,156.661
C00682=1048.914,129.058,-87.088,170.892,35.436,156.661
C00683=1048.920,129.307,-87.108,170.894,35.437,156.662
C00684=1048.926,129.555,-87.129,170.896,35.439,156.662
C00685=1048.932,129.805,-87.149,170.897,35.441,156.662
C00686=1048.938,130.054,-87.169,170.899,35.443,156.663
C00687=1048.944,130.303,-87.191,170.901,35.445,156.663
C00688=1048.951,130.553,-87.211,170.903,35.447,156.663
C00689=1048.957,130.801,-87.232,170.905,35.449,156.664
C00690=1048.963,131.051,-87.253,170.907,35.450,156.664
C00691=1048.970,131.299,-87.274,170.909,35.452,156.664
C00692=1048.975,131.549,-87.295,170.911,35.454,156.665
C00693=1048.982,131.798,-87.316,170.912,35.456,156.665
C00694=1048.988,132.047,-87.336,170.914,35.458,156.665
C00695=1048.994,132.296,-87.358,170.916,35.460,156.666
C00696=1049.000,132.544,-87.378,170.919,35.462,156.666
C00697=1049.006,132.794,-87.399,170.920,35.464,156.666
C00698=1049.011,133.042,-87.421,170.922,35.466,156.667
C00699=1049.018,133.292,-87.441,170.924,35.467,156.667
C00700=1049.024,133.541,-87.463,170.926,35.469,156.667
C00701=1049.030,133.790,-87.484,170.927,35.471,156.668
C00702=1049.036,134.039,-87.504,170.929,35.474,156.668
C00703=1049.042,134.288,-87.526,170.932,35.476,156.669
C00704=1049.048,134.537,-87.547,170.934,35.477,156.669
C00705=1049.054,134.786,-87.567,170.935,35.479,156.669
C00706=1049.060,135.035,-87.589,170.937,35.481,156.670
C00707=1049.066,135.284,-87.610,170.939,35.483,156.670
C00708=1049.072,135.533,-87.630,170.941,35.485,156.670
C00709=1049.079,135.782,-87.652,170.944,35.487,156.671
C00710=1049.085,136.031,-87.674,170.945,35.489,156.671
C00711=1049.091,136.280,-87.694,170.947,35.491,156.671
C00712=1049.097,136.529,-87.715,170.949,35.493,156.672
C00713=1049.102,136.778,-87.736,170.951,35.494,156.672
C00714=1049.109,137.027,-87.758,170.952,35.496,156.672
C00715=1049.115,137.277,-87.778,170.954,35.498,156.673
C00716=1049.121,137.525,-87.800,170.957,35.500,156.673
C00717=1049.127,137.774,-87.821,170.959,35.502,156.674
C00718=1049.133,138.024,-87.843,170.961,35.504,156.674
C00719=1049.139,138.272,-87.863,170.962,35.506,156.674
C00720=1049.145,138.522,-87.885,170.964,35.508,156.675
C00721=1049.151,138.771,-87.906,170.966,35.510,156.675
C00722=1049.157,139.019,-87.927,170.969,35.512,156.675
C00723=1049.164,139.268,-87.949,170.970,35.514,156.676
C00724=1049.170,139.518,-87.969,170.972,35.516,156.676
C00725=1049.175,139.766,-87.991,170.974,35.518,156.676
C00726=1049.181,140.016,-88.012,170.976,35.520,156.677
C00727=1049.188,140.265,-88.034,170.978,35.521,156.677
C00728=1049.193,140.513,-88.055,170.979,35.524,156.678
C00729=1049.199,140.763,-88.077,170.982,35.526,156.678
C00730=1049.205,141.012,-88.099,170.984,35.528,156.678
C00731=1049.212,141.260,-88.119,170.986,35.530,156.679
C00732=1049.219,141.546,-88.144,170.988,35.532,156.679
C00733=1049.225,141.831,-88.169,170.990,35.534,156.679
C00734=1049.232,142.117,-88.192,170.993,35.536,156.680
C00735=1049.239,142.403,-88.218,170.995,35.539,156.680
C00736=1049.246,142.652,-88.239,170.997,35.541,156.681
C00737=1049.251,142.900,-88.261,170.999,35.543,156.681
C00738=1049.257,143.150,-88.282,171.000,35.545,156.681
C00739=1049.263,143.399,-88.304,171.002,35.546,156.682
C00740=1049.269,143.647,-88.325,171.004,35.548,156.682
C00741=1049.275,143.896,-88.347,171.007,35.550,156.682
C00742=1049.281,144.146,-88.368,171.009,35.553,156.683
C00743=1049.287,144.395,-88.390,171.010,35.555,156.683
C00744=1049.293,144.643,-88.411,171.012,35.557,156.684
C00745=1049.299,144.893,-88.433,171.014,35.558,156.684
C00746=1049.305,145.142,-88.455,171.016,35.560,156.684
C00747=1049.312,145.391,-88.476,171.019,35.562,156.685
C00748=1049.318,145.639,-88.497,171.021,35.564,156.685
C00749=1049.324,145.888,-88.519,171.022,35.567,156.685
C00750=1049.330,146.138,-88.540,171.024,35.568,156.686
C00751=1049.336,146.387,-88.562,171.026,35.570,156.686
C00752=1049.343,146.635,-88.584,171.028,35.572,156.687
C00753=1049.348,146.884,-88.605,171.031,35.574,156.687
C00754=1049.355,147.133,-88.627,171.033,35.576,156.687
C00755=1049.361,147.382,-88.649,171.034,35.578,156.688
C00756=1049.367,147.632,-88.670,171.036,35.580,156.688
C00757=1049.373,147.881,-88.692,171.038,35.582,156.688
C00758=1049.378,148.130,-88.714,171.040,35.584,156.689
C00759=1049.384,148.378,-88.736,171.043,35.586,156.689
C00760=1049.390,148.627,-88.758,171.045,35.588,156.689
C00761=1049.397,148.877,-88.780,171.046,35.590,156.690
C00762=1049.403,149.126,-88.801,171.048,35.592,156.690
C00763=1049.408,149.374,-88.822,171.050,35.594,156.691
C00764=1049.415,149.623,-88.845,171.052,35.596,156.691
C00765=1049.421,149.872,-88.866,171.055,35.598,156.691
C00766=1049.426,150.122,-88.889,171.057,35.600,156.692
C00767=1049.433,150.371,-88.910,171.058,35.602,156.692
C00768=1049.438,150.619,-88.932,171.060,35.604,156.692
C00769=1049.445,150.868,-88.954,171.062,35.607,156.693
C00770=1049.451,151.117,-88.976,171.064,35.608,156.693
C00771=1049.456,151.366,-88.998,171.067,35.610,156.694
C00772=1049.463,151.615,-89.020,171.069,35.612,156.694
C00773=1049.469,151.864,-89.042,171.071,35.615,156.694
C00774=1049.475,152.113,-89.064,171.072,35.617,156.695
C00775=1049.481,152.361,-89.085,171.074,35.618,156.695
C00776=1049.486,152.611,-89.108,171.076,35.620,156.696
C00777=1049.493,152.860,-89.130,171.079,35.623,156.696
C00778=1049.499,153.109,-89.152,171.081,35.625,156.696
C00779=1049.505,153.358,-89.173,171.083,35.627,156.697
C00780=1049.511,153.607,-89.196,171.085,35.628,156.697
C00781=1049.517,153.856,-89.218,171.087,35.631,156.698
C00782=1049.523,154.105,-89.240,171.089,35.633,156.698
C00783=1049.529,154.353,-89.261,171.091,35.635,156.698
C00784=1049.534,154.603,-89.284,171.093,35.636,156.699
C00785=1049.541,154.851,-89.306,171.095,35.639,156.699
C00786=1049.547,155.100,-89.328,171.097,35.641,156.699
C00787=1049.554,155.349,-89.350,171.099,35.643,156.700
C00788=1049.559,155.599,-89.372,171.102,35.645,156.700
C00789=1049.565,155.847,-89.395,171.104,35.647,156.701
C00790=1049.571,156.097,-89.417,171.105,35.649,156.701
C00791=1049.577,156.345,-89.439,171.107,35.651,156.701
C00792=1049.583,156.594,-89.461,171.109,35.653,156.702
C00793=1049.589,156.843,-89.484,171.111,35.655,156.702
C00794=1049.595,157.092,-89.505,171.114,35.657,156.702
C00795=1049.601,157.340,-89.527,171.116,35.660,156.703
C00796=1049.608,157.626,-89.553,171.118,35.661,156.703
C00797=1049.615,157.911,-89.579,171.120,35.664,156.704
C00798=1049.622,158.197,-89.604,171.122,35.666,156.704
C00799=1049.629,158.481,-89.630,171.126,35.669,156.705
C00800=1049.635,158.730,-89.652,171.127,35.671,156.705
C00801=1049.641,158.979,-89.675,171.129,35.673,156.705
C00802=1049.647,159.229,-89.696,171.131,35.675,156.706
C00803=1049.653,159.477,-89.719,171.133,35.677,156.706
C00804=1049.659,159.726,-89.741,171.136,35.679,156.707
C00805=1049.665,159.975,-89.763,171.138,35.681,156.707
C00806=1049.672,160.224,-89.785,171.140,35.683,156.707
C00807=1049.677,160.473,-89.808,171.142,35.685,156.708
C00808=1049.683,160.722,-89.830,171.144,35.688,156.708
C00809=1049.689,160.971,-89.853,171.146,35.689,156.709
C00810=1049.695,161.220,-89.876,171.149,35.692,156.709
C00811=1049.701,161.469,-89.899,171.150,35.694,156.709
C00812=1049.706,161.718,-89.921,171.152,35.696,156.710
C00813=1049.712,161.967,-89.943,171.154,35.698,156.710
C00814=1049.718,162.216,-89.966,171.156,35.701,156.711
C00815=1049.724,162.465,-89.989,171.159,35.702,156.711
C00816=1049.729,162.714,-90.012,171.161,35.705,156.711
C00817=1049.736,162.963,-90.034,171.163,35.707,156.712
C00818=1049.742,163.212,-90.057,171.165,35.709,156.712
C00819=1049.747,163.460,-90.080,171.167,35.711,156.713
C00820=1049.753,163.709,-90.103,171.170,35.714,156.713
C00821=1049.759,163.957,-90.125,171.171,35.716,156.714
C00822=1049.765,164.206,-90.148,171.173,35.718,156.714
C00823=1049.770,164.456,-90.170,171.175,35.720,156.714
C00824=1049.776,164.705,-90.193,171.177,35.722,156.715
C00825=1049.782,164.953,-90.216,171.180,35.725,156.715
C00826=1049.788,165.202,-90.238,171.182,35.727,156.716
C00827=1049.794,165.451,-90.261,171.184,35.729,156.716
C00828=1049.799,165.700,-90.284,171.186,35.731,156.716
C00829=1049.806,165.949,-90.307,171.188,35.733,156.717
C00830=1049.812,166.198,-90.330,171.191,35.735,156.717
C00831=1049.818,166.447,-90.353,171.193,35.738,156.718
C00832=1049.824,166.696,-90.376,171.195,35.740,156.718
C00833=1049.829,166.945,-90.399,171.197,35.742,156.719
C00834=1049.835,167.194,-90.422,171.199,35.744,156.719
C00835=1049.841,167.442,-90.444,171.202,35.746,156.719
C00836=1049.847,167.691,-90.467,171.203,35.748,156.720
C00837=1049.853,167.940,-90.490,171.205,35.751,156.720
C00838=1049.859,168.189,-90.513,171.207,35.753,156.721
C00839=1049.865,168.438,-90.536,171.209,35.755,156.721
C00840=1049.870,168.687,-90.559,171.212,35.757,156.721
C00841=1049.877,168.935,-90.581,171.214,35.759,156.722
C00842=1049.882,169.184,-90.604,171.216,35.762,156.722
C00843=1049.888,169.433,-90.627,171.218,35.764,156.723
C00844=1049.895,169.683,-90.650,171.220,35.766,156.723
C00845=1049.900,169.932,-90.673,171.223,35.768,156.724
C00846=1049.906,170.180,-90.696,171.225,35.771,156.724
C00847=1049.912,170.429,-90.718,171.227,35.772,156.724
C00848=1049.918,170.678,-90.741,171.229,35.775,156.725
C00849=1049.924,170.926,-90.765,171.231,35.777,156.725
C00850=1049.930,171.175,-90.788,171.234,35.779,156.726
C00851=1049.936,171.425,-90.811,171.236,35.781,156.726
C00852=1049.942,171.674,-90.834,171.238,35.784,156.726
C00853=1049.949,171.922,-90.857,171.240,35.785,156.727
C00854=1049.954,172.171,-90.879,171.242,35.788,156.727
C00855=1049.960,172.419,-90.903,171.245,35.790,156.728
C00856=1049.966,172.668,-90.926,171.247,35.792,156.728
C00857=1049.972,172.918,-90.949,171.249,35.795,156.729
C00858=1049.978,173.167,-90.972,171.251,35.797,156.729
C00859=1049.984,173.416,-90.995,171.253,35.799,156.729
C00860=1049.991,173.699,-91.022,171.256,35.802,156.730
C00861=1049.998,173.985,-91.048,171.259,35.804,156.730
C00862=1050.005,174.269,-91.075,171.261,35.807,156.731
C00863=1050.012,174.554,-91.101,171.263,35.809,156.731
C00864=1050.017,174.803,-91.124,171.265,35.811,156.732
C00865=1050.024,175.052,-91.147,171.268,35.813,156.732
C00866=1050.031,175.301,-91.171,171.270,35.816,156.733
C00867=1050.036,175.550,-91.194,171.272,35.818,156.733
C00868=1050.042,175.798,-91.217,171.274,35.820,156.733
C00869=1050.048,176.047,-91.240,171.277,35.822,156.734
C00870=1050.054,176.296,-91.264,171.280,35.824,156.734
C00871=1050.060,176.545,-91.287,171.282,35.826,156.735
C00872=1050.066,176.794,-91.310,171.284,35.829,156.735
C00873=1050.072,177.042,-91.333,171.286,35.831,156.735
C00874=1050.079,177.292,-91.356,171.289,35.833,156.736
C00875=1050.085,177.540,-91.380,171.291,35.836,156.736
C00876=1050.091,177.789,-91.402,171.293,35.837,156.737
C00877=1050.097,178.038,-91.426,171.295,35.840,156.737
C00878=1050.103,178.287,-91.449,171.297,35.842,156.738
C00879=1050.109,178.536,-91.472,171.300,35.844,156.738
C00880=1050.115,178.785,-91.496,171.302,35.846,156.738
C00881=1050.121,179.034,-91.519,171.304,35.849,156.739
C00882=1050.127,179.282,-91.543,171.306,35.850,156.739
C00883=1050.134,179.531,-91.566,171.308,35.853,156.740
C00884=1050.140,179.779,-91.589,171.311,35.855,156.740
C00885=1050.146,180.028,-91.612,171.313,35.857,156.741
C00886=1050.153,180.277,-91.636,171.316,35.860,156.741
C00887=1050.158,180.526,-91.659,171.318,35.861,156.741
C00888=1050.165,180.775,-91.683,171.320,35.864,156.742
C00889=1050.171,181.024,-91.706,171.323,35.866,156.742
C00890=1050.177,181.272,-91.730,171.325,35.868,156.743
C00891=1050.183,181.522,-91.753,171.327,35.871,156.743
C00892=1050.189,181.770,-91.777,171.329,35.873,156.744
C00893=1050.196,182.020,-91.800,171.332,35.875,156.744
C00894=1050.202,182.268,-91.824,171.334,35.877,156.744
C00895=1050.208,182.516,-91.848,171.336,35.879,156.745
C00896=1050.214,182.766,-91.871,171.339,35.882,156.745
C00897=1050.220,183.014,-91.895,171.341,35.884,156.746
C00898=1050.226,183.264,-91.918,171.344,35.886,156.746
C00899=1050.233,183.512,-91.941,171.346,35.888,156.747
C00900=1050.240,183.761,-91.965,171.348,35.890,156.747
C00901=1050.245,184.010,-91.988,171.350,35.893,156.748
C00902=1050.251,184.258,-92.012,171.352,35.895,156.748
C00903=1050.257,184.507,-92.036,171.355,35.897,156.748
C00904=1050.262,184.756,-92.060,171.357,35.900,156.749
C00905=1050.268,185.005,-92.083,171.359,35.902,156.749
C00906=1050.274,185.254,-92.108,171.361,35.905,156.750
C00907=1050.280,185.502,-92.132,171.365,35.907,156.750
C00908=1050.286,185.751,-92.156,171.367,35.909,156.751
C00909=1050.292,186.000,-92.179,171.369,35.912,156.751
C00910=1050.298,186.249,-92.203,171.371,35.914,156.752
C00911=1050.304,186.498,-92.227,171.374,35.916,156.752
C00912=1050.310,186.746,-92.251,171.376,35.919,156.753
C00913=1050.315,186.995,-92.275,171.378,35.921,156.753
C00914=1050.322,187.244,-92.299,171.380,35.924,156.753
C00915=1050.327,187.492,-92.324,171.383,35.926,156.754
C00916=1050.333,187.741,-92.347,171.385,35.929,156.754
C00917=1050.339,187.991,-92.371,171.388,35.931,156.755
C00918=1050.345,188.239,-92.395,171.390,35.933,156.755
C00919=1050.351,188.488,-92.420,171.392,35.936,156.756
C00920=1050.357,188.736,-92.443,171.395,35.938,156.756
C00921=1050.363,188.986,-92.468,171.397,35.941,156.757
C00922=1050.369,189.234,-92.491,171.399,35.943,156.757
C00923=1050.374,189.483,-92.516,171.401,35.945,156.758
C00924=1050.381,189.767,-92.543,171.405,35.948,156.758
C00925=1050.388,190.052,-92.571,171.407,35.951,156.759
C00926=1050.395,190.336,-92.598,171.410,35.954,156.759
C00927=1050.402,190.620,-92.626,171.413,35.956,156.760
C00928=1050.408,190.869,-92.650,171.415,35.959,156.760
C00929=1050.414,191.118,-92.675,171.417,35.961,156.761
C00930=1050.419,191.366,-92.699,171.420,35.963,156.761
C00931=1050.426,191.615,-92.723,171.422,35.966,156.762
C00932=1050.431,191.864,-92.747,171.425,35.968,156.762
C00933=1050.438,192.113,-92.771,171.427,35.971,156.763
C00934=1050.443,192.361,-92.795,171.429,35.973,156.763
C00935=1050.450,192.610,-92.819,171.431,35.976,156.764
C00936=1050.455,192.859,-92.844,171.435,35.978,156.764
C00937=1050.462,193.108,-92.868,171.437,35.981,156.765
C00938=1050.467,193.356,-92.892,171.439,35.983,156.765
C00939=1050.474,193.605,-92.917,171.441,35.986,156.766
C00940=1050.479,193.853,-92.941,171.444,35.988,156.766
C00941=1050.485,194.103,-92.966,171.446,35.990,156.767
C00942=1050.492,194.352,-92.990,171.449,35.993,156.767
C00943=1050.497,194.600,-93.014,171.451,35.995,156.768
C00944=1050.504,194.849,-93.038,171.454,35.998,156.768
C00945=1050.510,195.097,-93.063,171.456,36.000,156.769
C00946=1050.516,195.346,-93.087,171.458,36.002,156.769
C00947=1050.522,195.595,-93.111,171.461,36.005,156.769
C00948=1050.528,195.844,-93.135,171.464,36.007,156.770
C00949=1050.534,196.092,-93.160,171.466,36.009,156.770
C00950=1050.540,196.341,-93.184,171.468,36.012,156.771
C00951=1050.546,196.590,-93.209,171.470,36.014,156.771
C00952=1050.552,196.839,-93.233,171.474,36.017,156.772
C00953=1050.558,197.087,-93.258,171.476,36.019,156.772
C00954=1050.564,197.336,-93.282,171.478,36.022,156.773
C00955=1050.571,197.585,-93.306,171.480,36.024,156.773
C00956=1050.577,197.833,-93.331,171.484,36.027,156.774
C00957=1050.583,198.082,-93.355,171.486,36.029,156.774
C00958=1050.589,198.331,-93.380,171.488,36.031,156.775
C00959=1050.595,198.579,-93.405,171.490,36.034,156.775
C00960=1050.601,198.828,-93.429,171.494,36.036,156.776
C00961=1050.607,199.078,-93.454,171.496,36.039,156.776
C00962=1050.614,199.325,-93.478,171.498,36.042,156.777
C00963=1050.620,199.575,-93.503,171.500,36.044,156.777
C00964=1050.625,199.824,-93.527,171.504,36.047,156.778
C00965=1050.632,200.072,-93.552,171.506,36.049,156.778
C00966=1050.638,200.321,-93.576,171.508,36.052,156.779
C00967=1050.645,200.569,-93.601,171.510,36.054,156.779
C00968=1050.651,200.818,-93.626,171.514,36.056,156.780
C00969=1050.657,201.067,-93.651,171.516,36.059,156.780
C00970=1050.663,201.315,-93.675,171.518,36.061,156.781
C00971=1050.669,201.564,-93.700,171.520,36.064,156.781
C00972=1050.675,201.813,-93.725,171.524,36.066,156.782
C00973=1050.681,202.062,-93.750,171.526,36.069,156.782
C00974=1050.687,202.310,-93.774,171.528,36.072,156.783
C00975=1050.693,202.559,-93.799,171.531,36.074,156.783
C00976=1050.699,202.808,-93.824,171.534,36.077,156.784
C00977=1050.705,203.056,-93.849,171.536,36.079,156.784
C00978=1050.711,203.305,-93.874,171.538,36.081,156.785
C00979=1050.717,203.554,-93.898,171.541,36.084,156.785
C00980=1050.723,203.803,-93.924,171.544,36.087,156.786
C00981=1050.729,204.051,-93.949,171.546,36.089,156.786
C00982=1050.735,204.300,-93.973,171.548,36.092,156.787
C00983=1050.741,204.549,-93.999,171.552,36.095,156.787
C00984=1050.747,204.797,-94.024,171.554,36.097,156.788
C00985=1050.752,205.046,-94.048,171.556,36.100,156.788
C00986=1050.759,205.294,-94.073,171.559,36.103,156.789
C00987=1050.766,205.543,-94.098,171.562,36.105,156.789
C00988=1050.790,206.596,-94.204,171.789,36.201,156.808
C00989=1050.797,206.846,-94.231,171.790,36.205,156.809
C00990=1050.804,207.098,-94.257,171.793,36.208,156.809
C00991=1050.810,207.349,-94.283,171.795,36.211,156.810
C00992=1050.817,207.600,-94.309,171.797,36.215,156.811
C00993=1050.824,207.849,-94.336,171.799,36.218,156.812
C00994=1050.829,208.098,-94.362,171.801,36.221,156.812
C00995=1050.836,208.346,-94.388,171.803,36.225,156.813
C00996=1050.843,208.594,-94.414,171.805,36.228,156.814
C00997=1050.849,208.843,-94.441,171.806,36.232,156.814
C00998=1050.855,209.092,-94.466,171.809,36.235,156.815
C00999=1050.862,209.340,-94.493,171.811,36.238,156.816
C01000=1050.869,209.588,-94.519,171.813,36.242,156.816
C01001=1050.874,209.837,-94.545,171.815,36.245,156.817
C01002=1050.881,210.086,-94.571,171.816,36.248,156.818
C01003=1050.888,210.334,-94.597,171.819,36.252,156.819
C01004=1050.893,210.582,-94.624,171.821,36.256,156.819
C01005=1050.901,210.831,-94.650,171.823,36.259,156.820
C01006=1050.906,211.080,-94.676,171.825,36.262,156.821
C01007=1050.913,211.329,-94.702,171.827,36.266,156.821
C01008=1050.920,211.577,-94.728,171.829,36.269,156.822
C01009=1050.925,211.825,-94.755,171.831,36.272,156.823
C01010=1050.933,212.074,-94.782,171.832,36.275,156.823
C01011=1050.938,212.322,-94.808,171.835,36.279,156.824
C01012=1050.945,212.570,-94.834,171.837,36.283,156.825
C01013=1050.951,212.820,-94.861,171.839,36.286,156.825
C01014=1050.957,213.068,-94.887,171.841,36.289,156.826
C01015=1050.964,213.317,-94.914,171.843,36.293,156.827
C01016=1050.970,213.565,-94.940,171.845,36.296,156.828
C01017=1050.976,213.814,-94.966,171.847,36.299,156.828
C01018=1050.983,214.062,-94.993,171.850,36.303,156.829
C01019=1050.989,214.311,-95.019,171.851,36.306,156.830
C01020=1050.996,214.560,-95.046,171.853,36.310,156.830
C01021=1051.002,214.808,-95.072,171.856,36.313,156.831
C01022=1051.008,215.056,-95.099,171.857,36.316,156.832
C01023=1051.015,215.305,-95.126,171.860,36.320,156.832
C01024=1051.021,215.553,-95.152,171.862,36.323,156.833
C01025=1051.028,215.802,-95.179,171.863,36.326,156.834
C01026=1051.033,216.050,-95.205,171.866,36.330,156.835
C01027=1051.041,216.299,-95.232,171.868,36.333,156.835
C01028=1051.046,216.548,-95.258,171.870,36.337,156.836
C01029=1051.053,216.796,-95.286,171.872,36.340,156.837
C01030=1051.059,217.044,-95.312,171.874,36.343,156.837
C01031=1051.066,217.293,-95.339,171.877,36.347,156.838
C01032=1051.072,217.541,-95.365,171.878,36.350,156.839
C01033=1051.079,217.790,-95.392,171.881,36.353,156.839
C01034=1051.085,218.038,-95.418,171.883,36.357,156.840
C01035=1051.092,218.287,-95.445,171.884,36.360,156.841
C01036=1051.097,218.536,-95.472,171.887,36.364,156.842
C01037=1051.105,218.784,-95.499,171.889,36.366,156.842
C01038=1051.111,219.032,-95.526,171.891,36.370,156.843
C01039=1051.118,219.281,-95.552,171.893,36.373,156.844
C01040=1051.123,219.529,-95.579,171.895,36.377,156.844
C01041=1051.130,219.778,-95.606,171.898,36.380,156.845
C01042=1051.136,220.026,-95.632,171.899,36.383,156.846
C01043=1051.143,220.275,-95.660,171.902,36.387,156.846
C01044=1051.150,220.523,-95.686,171.904,36.390,156.847
C01045=1051.156,220.780,-95.714,171.906,36.393,156.848
C01046=1051.163,221.037,-95.742,171.908,36.397,156.848
C01047=1051.169,221.294,-95.769,171.910,36.400,156.849
C01048=1051.176,221.550,-95.797,171.913,36.404,156.850
C01049=1051.182,221.798,-95.824,171.915,36.407,156.851
C01050=1051.189,222.047,-95.851,171.917,36.410,156.851
C01051=1051.194,222.296,-95.878,171.919,36.414,156.852
C01052=1051.201,222.544,-95.906,171.921,36.417,156.853
C01053=1051.207,222.792,-95.932,171.924,36.420,156.853
C01054=1051.213,223.041,-95.959,171.926,36.424,156.854
C01055=1051.221,223.290,-95.986,171.927,36.427,156.855
C01056=1051.226,223.538,-96.013,171.930,36.430,156.855
C01057=1051.233,223.786,-96.041,171.932,36.434,156.856
C01058=1051.239,224.035,-96.067,171.935,36.437,156.857
C01059=1051.245,224.283,-96.095,171.936,36.441,156.858
C01060=1051.252,224.532,-96.122,171.938,36.444,156.858
C01061=1051.258,224.780,-96.148,171.941,36.447,156.859
C01062=1051.265,225.029,-96.176,171.943,36.451,156.860
C01063=1051.271,225.277,-96.203,171.945,36.454,156.860
C01064=1051.278,225.526,-96.230,171.947,36.457,156.861
C01065=1051.284,225.775,-96.257,171.949,36.460,156.862
C01066=1051.290,226.022,-96.285,171.952,36.464,156.862
C01067=1051.296,226.271,-96.312,171.954,36.467,156.863
C01068=1051.303,226.520,-96.339,171.956,36.470,156.864
C01069=1051.310,226.768,-96.366,171.958,36.473,156.864
C01070=1051.316,227.016,-96.393,171.961,36.477,156.865
C01071=1051.323,227.265,-96.421,171.963,36.480,156.866
C01072=1051.329,227.513,-96.448,171.965,36.484,156.867
C01073=1051.335,227.762,-96.475,171.968,36.487,156.867
C01074=1051.342,228.011,-96.502,171.969,36.490,156.868
C01075=1051.348,228.258,-96.530,171.972,36.493,156.869
C01076=1051.354,228.507,-96.557,171.974,36.497,156.869
C01077=1051.361,228.756,-96.584,171.976,36.500,156.870
C01078=1051.368,229.004,-96.612,171.979,36.503,156.871
C01079=1051.373,229.253,-96.639,171.980,36.506,156.871
C01080=1051.380,229.501,-96.667,171.983,36.510,156.872
C01081=1051.387,229.750,-96.694,171.985,36.513,156.873
C01082=1051.393,229.997,-96.722,171.987,36.516,156.873
C01083=1051.399,230.246,-96.749,171.990,36.520,156.874
C01084=1051.406,230.495,-96.776,171.992,36.523,156.875
C01085=1051.412,230.743,-96.804,171.994,36.526,156.875
C01086=1051.419,230.991,-96.832,171.996,36.529,156.876
C01087=1051.425,231.240,-96.859,171.999,36.533,156.877
C01088=1051.430,231.488,-96.886,172.001,36.536,156.877
C01089=1051.437,231.737,-96.914,172.003,36.540,156.878
C01090=1051.444,231.985,-96.942,172.006,36.543,156.879
C01091=1051.450,232.233,-96.970,172.008,36.546,156.880
C01092=1051.456,232.482,-96.996,172.010,36.550,156.880
C01093=1051.463,232.730,-97.024,172.012,36.553,156.881
C01094=1051.469,232.979,-97.052,172.014,36.556,156.882
C01095=1051.475,233.227,-97.080,172.017,36.559,156.882
C01096=1051.481,233.475,-97.107,172.019,36.563,156.883
C01097=1051.488,233.724,-97.135,172.022,36.566,156.884
C01098=1051.495,233.972,-97.163,172.024,36.569,156.885
C01099=1051.501,234.221,-97.191,172.027,36.573,156.885
C01100=1051.507,234.469,-97.219,172.028,36.576,156.886
C01101=1051.514,234.718,-97.246,172.030,36.579,156.887
C01102=1051.520,234.967,-97.274,172.033,36.582,156.887
C01103=1051.526,235.216,-97.301,172.035,36.586,156.888
C01104=1051.533,235.466,-97.330,172.038,36.589,156.889
C01105=1051.539,235.714,-97.358,172.040,36.592,156.889
C01106=1051.545,235.962,-97.386,172.043,36.596,156.890
C01107=1051.551,236.211,-97.413,172.045,36.599,156.891
C01108=1051.558,236.459,-97.441,172.047,36.603,156.892
C01109=1051.565,236.707,-97.469,172.049,36.606,156.892
C01110=1051.571,236.956,-97.497,172.051,36.609,156.893
C01111=1051.577,237.205,-97.525,172.054,36.612,156.894
C01112=1051.583,237.452,-97.552,172.056,36.616,156.894
C01113=1051.589,237.701,-97.581,172.058,36.619,156.895
C01114=1051.596,237.950,-97.608,172.061,36.622,156.896
C01115=1051.603,238.198,-97.636,172.063,36.625,156.896
C01116=1051.609,238.446,-97.664,172.066,36.629,156.897
C01117=1051.616,238.695,-97.693,172.068,36.632,156.898
C01118=1051.622,238.943,-97.721,172.071,36.635,156.898
C01119=1051.628,239.191,-97.748,172.073,36.638,156.899
C01120=1051.634,239.439,-97.776,172.075,36.642,156.900
C01121=1051.641,239.688,-97.804,172.078,36.645,156.900
C01122=1051.648,239.936,-97.832,172.080,36.648,156.901
C01123=1051.654,240.185,-97.861,172.083,36.651,156.902
C01124=1051.661,240.433,-97.889,172.085,36.655,156.903
C01125=1051.667,240.682,-97.917,172.088,36.658,156.903
C01126=1051.673,240.930,-97.945,172.089,36.661,156.904
C01127=1051.680,241.178,-97.973,172.091,36.664,156.905
C01128=1051.686,241.427,-98.001,172.094,36.668,156.905
C01129=1051.693,241.675,-98.029,172.096,36.671,156.906
C01130=1051.698,241.923,-98.057,172.099,36.674,156.907
C01131=1051.705,242.171,-98.085,172.101,36.677,156.907
C01132=1051.711,242.420,-98.114,172.104,36.681,156.908
C01133=1051.718,242.668,-98.142,172.106,36.684,156.909
C01134=1051.724,242.916,-98.171,172.108,36.687,156.910
C01135=1051.730,243.165,-98.199,172.111,36.691,156.910
C01136=1051.737,243.413,-98.227,172.113,36.694,156.911
C01137=1051.743,243.662,-98.256,172.116,36.697,156.912
C01138=1051.750,243.910,-98.283,172.118,36.700,156.912
C01139=1051.756,244.158,-98.312,172.121,36.704,156.913
C01140=1051.763,244.407,-98.340,172.123,36.707,156.914
C01141=1051.769,244.655,-98.369,172.126,36.710,156.914
C01142=1051.775,244.904,-98.398,172.128,36.714,156.915
C01143=1051.782,245.151,-98.426,172.130,36.717,156.916
C01144=1051.788,245.400,-98.454,172.133,36.720,156.917
C01145=1051.794,245.648,-98.483,172.135,36.723,156.917
C01146=1051.801,245.897,-98.511,172.138,36.727,156.918
C01147=1051.807,246.145,-98.540,172.140,36.730,156.919
C01148=1051.812,246.393,-98.568,172.143,36.733,156.919
C01149=1051.819,246.641,-98.597,172.145,36.737,156.920
C01150=1051.826,246.889,-98.626,172.147,36.740,156.921
C01151=1051.831,247.138,-98.654,172.150,36.743,156.922
C01152=1051.838,247.386,-98.683,172.152,36.747,156.922
C01153=1051.844,247.634,-98.711,172.155,36.750,156.923
C01154=1051.850,247.883,-98.740,172.157,36.754,156.924
C01155=1051.856,248.131,-98.769,172.160,36.757,156.924
C01156=1051.862,248.380,-98.798,172.162,36.760,156.925
C01157=1051.868,248.625,-98.826,172.165,36.764,156.926
C01158=1051.875,248.870,-98.855,172.167,36.767,156.926
C01159=1051.881,249.116,-98.883,172.170,36.770,156.927
C01160=1051.888,249.362,-98.912,172.172,36.773,156.928
C01161=1051.894,249.608,-98.940,172.174,36.777,156.929
C01162=1051.900,249.854,-98.969,172.177,36.780,156.929
C01163=1051.906,250.100,-98.997,172.179,36.783,156.930
C01164=1051.913,250.345,-99.026,172.182,36.787,156.931
C01165=1051.919,250.594,-99.055,172.184,36.790,156.931
C01166=1051.925,250.842,-99.084,172.188,36.793,156.932
C01167=1051.931,251.090,-99.112,172.190,36.796,156.933
C01168=1051.937,251.339,-99.141,172.193,36.800,156.934
C01169=1051.943,251.587,-99.170,172.195,36.803,156.934
C01170=1051.950,251.834,-99.199,172.197,36.806,156.935
C01171=1051.957,252.083,-99.228,172.200,36.810,156.936
C01172=1051.964,252.331,-99.257,172.202,36.813,156.936
C01173=1051.970,252.580,-99.286,172.205,36.816,156.937
C01174=1051.976,252.828,-99.314,172.207,36.819,156.938
C01175=1051.982,253.076,-99.343,172.210,36.823,156.938
C01176=1051.988,253.325,-99.372,172.212,36.826,156.939
C01177=1051.994,253.573,-99.401,172.215,36.829,156.940
C01178=1052.001,253.821,-99.430,172.218,36.833,156.941
C01179=1052.007,254.069,-99.460,172.221,36.835,156.941
C01180=1052.015,254.318,-99.488,172.223,36.839,156.942
C01181=1052.021,254.566,-99.517,172.225,36.842,156.943
C01182=1052.027,254.814,-99.546,172.228,36.845,156.943
C01183=1052.033,255.062,-99.575,172.230,36.849,156.944
C01184=1052.040,255.310,-99.604,172.233,36.852,156.945
C01185=1052.046,255.558,-99.634,172.235,36.855,156.946
C01186=1052.053,255.807,-99.663,172.239,36.858,156.946
C01187=1052.059,256.055,-99.692,172.241,36.862,156.947
C01188=1052.065,256.303,-99.721,172.244,36.865,156.948
C01189=1052.071,256.551,-99.750,172.246,36.868,156.948
C01190=1052.078,256.800,-99.779,172.249,36.871,156.949
C01191=1052.085,257.048,-99.809,172.251,36.875,156.950
C01192=1052.091,257.297,-99.838,172.253,36.878,156.950
C01193=1052.098,257.544,-99.867,172.257,36.881,156.951
C01194=1052.104,257.792,-99.896,172.259,36.884,156.952
C01195=1052.111,258.041,-99.925,172.262,36.888,156.953
C01196=1052.117,258.289,-99.954,172.264,36.891,156.953
C01197=1052.124,258.537,-99.983,172.267,36.894,156.954
C01198=1052.131,258.786,-100.013,172.269,36.898,156.955
C01199=1052.137,259.034,-100.042,172.273,36.901,156.955
C01200=1052.143,259.281,-100.071,172.275,36.904,156.956
C01201=1052.150,259.530,-100.100,172.278,36.907,156.957
C01202=1052.156,259.778,-100.130,172.280,36.911,156.958
C01203=1052.163,260.026,-100.159,172.283,36.914,156.958
C01204=1052.169,260.274,-100.189,172.286,36.917,156.959
C01205=1052.176,260.523,-100.218,172.288,36.920,156.960
C01206=1052.182,260.771,-100.247,172.291,36.924,156.960
C01207=1052.189,261.019,-100.276,172.293,36.927,156.961
C01208=1052.196,261.267,-100.306,172.296,36.930,156.962
C01209=1052.202,261.515,-100.335,172.299,36.933,156.962
C01210=1052.208,261.764,-100.364,172.302,36.936,156.963
C01211=1052.215,262.012,-100.395,172.304,36.939,156.964
C01212=1052.222,262.260,-100.424,172.307,36.943,156.965
C01213=1052.228,262.505,-100.453,172.310,36.946,156.965
C01214=1052.235,262.750,-100.481,172.313,36.949,156.966
C01215=1052.242,262.995,-100.510,172.315,36.952,156.967
C01216=1052.248,263.240,-100.541,172.318,36.956,156.967
C01217=1052.253,263.484,-100.570,172.320,36.959,156.968
C01218=1052.260,263.729,-100.599,172.324,36.962,156.969
C01219=1052.266,263.975,-100.628,172.326,36.965,156.970
C01220=1052.273,264.219,-100.658,172.328,36.969,156.970
C01221=1052.279,264.467,-100.687,172.331,36.972,156.971
C01222=1052.285,264.715,-100.717,172.333,36.975,156.972
C01223=1052.292,264.964,-100.747,172.337,36.979,156.972
C01224=1052.298,265.211,-100.776,172.339,36.982,156.973
C01225=1052.304,265.460,-100.806,172.342,36.985,156.974
C01226=1052.311,265.708,-100.836,172.344,36.989,156.975
C01227=1052.318,265.956,-100.866,172.348,36.992,156.975
C01228=1052.324,266.205,-100.896,172.350,36.995,156.976
C01229=1052.330,266.452,-100.926,172.353,36.999,156.977
C01230=1052.337,266.700,-100.955,172.355,37.002,156.978
C01231=1052.343,266.949,-100.985,172.359,37.005,156.978
C01232=1052.349,267.196,-101.015,172.361,37.008,156.979
C01233=1052.357,267.445,-101.045,172.364,37.012,156.980
C01234=1052.362,267.693,-101.075,172.366,37.015,156.980
C01235=1052.369,267.941,-101.105,172.370,37.018,156.981
C01236=1052.375,268.189,-101.135,172.372,37.021,156.982
C01237=1052.381,268.437,-101.164,172.375,37.025,156.983
C01238=1052.388,268.686,-101.195,172.378,37.028,156.983
C01239=1052.394,268.933,-101.225,172.381,37.032,156.984
C01240=1052.401,269.182,-101.256,172.383,37.035,156.985
C01241=1052.407,269.429,-101.285,172.386,37.038,156.986
C01242=1052.414,269.678,-101.315,172.389,37.042,156.986
C01243=1052.420,269.926,-101.345,172.392,37.045,156.987
C01244=1052.427,270.174,-101.375,172.394,37.048,156.988
C01245=1052.433,270.422,-101.406,172.398,37.052,156.989
C01246=1052.439,270.670,-101.436,172.400,37.055,156.989
C01247=1052.446,270.918,-101.466,172.403,37.058,156.990
C01248=1052.452,271.166,-101.497,172.406,37.062,156.991
C01249=1052.459,271.415,-101.526,172.409,37.065,156.991
C01250=1052.465,271.663,-101.556,172.411,37.068,156.992
C01251=1052.472,271.911,-101.586,172.415,37.071,156.993
C01252=1052.478,272.159,-101.617,172.417,37.075,156.994
C01253=1052.485,272.407,-101.647,172.420,37.078,156.994
C01254=1052.491,272.655,-101.677,172.423,37.081,156.995
C01255=1052.497,272.903,-101.708,172.426,37.085,156.996
C01256=1052.504,273.151,-101.738,172.428,37.088,156.997
C01257=1052.510,273.399,-101.768,172.432,37.091,156.997
C01258=1052.516,273.648,-101.799,172.434,37.095,156.998
C01259=1052.523,273.894,-101.829,172.437,37.098,156.999
C01260=1052.529,274.143,-101.860,172.440,37.102,157.000
C01261=1052.535,274.391,-101.891,172.443,37.105,157.000
C01262=1052.542,274.639,-101.921,172.445,37.108,157.001
C01263=1052.549,274.888,-101.951,172.449,37.112,157.002
C01264=1052.555,275.135,-101.982,172.451,37.115,157.003
C01265=1052.562,275.384,-102.012,172.454,37.119,157.003
C01266=1052.568,275.631,-102.042,172.457,37.122,157.004
C01267=1052.574,275.879,-102.074,172.460,37.125,157.005
C01268=1052.580,276.127,-102.104,172.463,37.128,157.006
C01269=1052.587,276.374,-102.134,172.466,37.132,157.006
C01270=1052.594,276.621,-102.164,172.468,37.135,157.007
C01271=1052.600,276.869,-102.195,172.472,37.138,157.008
C01272=1052.606,277.115,-102.225,172.474,37.142,157.009
C01273=1052.613,277.362,-102.256,172.477,37.145,157.009
C01274=1052.619,277.609,-102.287,172.480,37.149,157.010
C01275=1052.626,277.856,-102.317,172.483,37.152,157.011
C01276=1052.633,278.103,-102.348,172.486,37.155,157.012
C01277=1052.639,278.350,-102.378,172.489,37.159,157.012
C01278=1052.645,278.599,-102.409,172.491,37.162,157.013
C01279=1052.652,278.847,-102.440,172.495,37.165,157.014
C01280=1052.658,279.095,-102.471,172.497,37.169,157.014
C01281=1052.665,279.343,-102.501,172.501,37.172,157.015
C01282=1052.671,279.591,-102.532,172.503,37.176,157.016
C01283=1052.677,279.839,-102.563,172.507,37.179,157.017
C01284=1052.684,280.087,-102.594,172.510,37.182,157.018
C01285=1052.690,280.335,-102.625,172.512,37.186,157.018
C01286=1052.696,280.582,-102.656,172.516,37.189,157.019
C01287=1052.703,280.831,-102.687,172.518,37.192,157.020
C01288=1052.710,281.079,-102.718,172.522,37.196,157.021
C01289=1052.715,281.327,-102.748,172.524,37.199,157.021
C01290=1052.722,281.574,-102.780,172.527,37.203,157.022
C01291=1052.729,281.823,-102.810,172.530,37.206,157.023
C01292=1052.735,282.070,-102.842,172.533,37.210,157.024
C01293=1052.741,282.319,-102.872,172.536,37.213,157.025
C01294=1052.748,282.567,-102.904,172.539,37.217,157.025
C01295=1052.754,282.814,-102.935,172.542,37.220,157.026
C01296=1052.760,283.062,-102.965,172.545,37.224,157.027
C01297=1052.767,283.310,-102.997,172.548,37.226,157.027
C01298=1052.774,283.558,-103.028,172.551,37.230,157.028
C01299=1052.780,283.806,-103.059,172.554,37.233,157.029
C01300=1052.786,284.054,-103.090,172.557,37.237,157.030
C01301=1052.793,284.302,-103.122,172.561,37.240,157.031
C01302=1052.800,284.550,-103.152,172.563,37.244,157.031
C01303=1052.806,284.799,-103.184,172.567,37.247,157.032
C01304=1052.812,285.046,-103.215,172.569,37.251,157.033
C01305=1052.818,285.294,-103.247,172.573,37.254,157.034
C01306=1052.825,285.542,-103.277,172.575,37.258,157.035
C01307=1052.832,285.790,-103.309,172.579,37.261,157.035
C01308=1052.838,286.038,-103.340,172.581,37.265,157.036
C01309=1052.845,286.286,-103.372,172.585,37.267,157.037
C01310=1052.851,286.533,-103.403,172.587,37.271,157.038
C01311=1052.857,286.782,-103.434,172.591,37.274,157.038
C01312=1052.864,287.029,-103.465,172.594,37.278,157.039
C01313=1052.871,287.277,-103.496,172.597,37.281,157.040
C01314=1052.878,287.525,-103.528,172.600,37.285,157.041
C01315=1052.884,287.773,-103.559,172.603,37.288,157.041
C01316=1052.891,288.021,-103.591,172.606,37.292,157.042
C01317=1052.897,288.269,-103.622,172.609,37.295,157.043
C01318=1052.903,288.516,-103.654,172.612,37.299,157.044
C01319=1052.910,288.764,-103.685,172.615,37.302,157.045
C01320=1052.917,289.012,-103.717,172.618,37.306,157.045
C01321=1052.923,289.261,-103.749,172.622,37.309,157.046
C01322=1052.929,289.508,-103.780,172.624,37.312,157.047
C01323=1052.936,289.756,-103.812,172.628,37.316,157.048
C01324=1052.943,290.004,-103.843,172.631,37.319,157.049
C01325=1052.949,290.262,-103.876,172.634,37.323,157.049
C01326=1052.956,290.519,-103.909,172.637,37.327,157.050
C01327=1052.962,290.776,-103.941,172.641,37.330,157.051
C01328=1052.970,291.032,-103.974,172.644,37.334,157.052
C01329=1052.976,291.281,-104.006,172.647,37.338,157.053
C01330=1052.982,291.529,-104.038,172.650,37.341,157.053
C01331=1052.989,291.776,-104.069,172.653,37.345,157.054
C01332=1052.995,292.025,-104.101,172.657,37.348,157.055
C01333=1053.002,292.273,-104.133,172.659,37.352,157.056
C01334=1053.009,292.520,-104.165,172.663,37.355,157.057
C01335=1053.014,292.767,-104.197,172.666,37.359,157.057
C01336=1053.021,293.015,-104.228,172.669,37.362,157.058
C01337=1053.027,293.263,-104.260,172.673,37.365,157.059
C01338=1053.034,293.511,-104.292,172.675,37.369,157.060
C01339=1053.041,293.759,-104.324,172.679,37.372,157.061
C01340=1053.047,294.007,-104.356,172.681,37.376,157.061
C01341=1053.054,294.254,-104.388,172.685,37.380,157.062
C01342=1053.060,294.502,-104.419,172.689,37.383,157.063
C01343=1053.067,294.751,-104.452,172.691,37.387,157.064
C01344=1053.074,294.998,-104.484,172.695,37.390,157.065
C01345=1053.080,295.246,-104.516,172.697,37.394,157.065
C01346=1053.087,295.494,-104.547,172.701,37.397,157.066
C01347=1053.093,295.742,-104.580,172.705,37.401,157.067
C01348=1053.100,295.990,-104.611,172.707,37.404,157.068
C01349=1053.106,296.237,-104.644,172.711,37.408,157.069
C01350=1053.113,296.485,-104.676,172.714,37.411,157.070
C01351=1053.119,296.733,-104.708,172.717,37.415,157.070
C01352=1053.125,296.981,-104.740,172.720,37.419,157.071
C01353=1053.131,297.229,-104.773,172.724,37.422,157.072
C01354=1053.138,297.476,-104.805,172.727,37.426,157.073
C01355=1053.144,297.724,-104.837,172.730,37.430,157.074
C01356=1053.151,297.972,-104.870,172.733,37.433,157.075
C01357=1053.157,298.220,-104.902,172.737,37.437,157.075
C01358=1053.163,298.468,-104.935,172.740,37.441,157.076
C01359=1053.170,298.715,-104.967,172.743,37.444,157.077
C01360=1053.176,298.963,-104.999,172.746,37.448,157.078
C01361=1053.182,299.211,-105.032,172.750,37.451,157.079
C01362=1053.188,299.458,-105.064,172.753,37.455,157.080
C01363=1053.194,299.707,-105.096,172.756,37.459,157.080
C01364=1053.202,299.954,-105.129,172.760,37.462,157.081
C01365=1053.208,300.201,-105.161,172.762,37.466,157.082
C01366=1053.215,300.450,-105.194,172.766,37.470,157.083
C01367=1053.221,300.697,-105.227,172.770,37.473,157.084
C01368=1053.227,300.946,-105.259,172.772,37.477,157.085
C01369=1053.234,301.193,-105.291,172.776,37.481,157.085
C01370=1053.240,301.440,-105.324,172.779,37.484,157.086
C01371=1053.247,301.688,-105.357,172.783,37.488,157.087
C01372=1053.253,301.936,-105.390,172.786,37.492,157.088
C01373=1053.260,302.184,-105.423,172.789,37.496,157.089
C01374=1053.266,302.432,-105.455,172.793,37.499,157.090
C01375=1053.273,302.679,-105.487,172.796,37.502,157.091
C01376=1053.279,302.927,-105.520,172.799,37.506,157.091
C01377=1053.285,303.175,-105.552,172.803,37.510,157.092
C01378=1053.292,303.422,-105.585,172.806,37.514,157.093
C01379=1053.299,303.670,-105.618,172.809,37.517,157.094
C01380=1053.305,303.918,-105.651,172.813,37.521,157.095
C01381=1053.312,304.191,-105.687,172.816,37.525,157.096
C01382=1053.320,304.464,-105.723,172.820,37.529,157.097
C01383=1053.327,304.737,-105.759,172.824,37.533,157.098
C01384=1053.334,305.010,-105.795,172.827,37.537,157.099
C01385=1053.341,305.258,-105.828,172.831,37.541,157.099
C01386=1053.347,305.505,-105.861,172.835,37.545,157.100
C01387=1053.353,305.753,-105.894,172.838,37.548,157.101
C01388=1053.361,306.001,-105.926,172.841,37.552,157.102
C01389=1053.367,306.248,-105.960,172.845,37.555,157.103
C01390=1053.374,306.496,-105.992,172.848,37.559,157.104
C01391=1053.381,306.744,-106.025,172.852,37.563,157.105
C01392=1053.387,306.991,-106.058,172.856,37.567,157.106
C01393=1053.393,307.239,-106.091,172.858,37.570,157.106
C01394=1053.400,307.487,-106.124,172.862,37.574,157.107
C01395=1053.407,307.734,-106.157,172.865,37.578,157.108
C01396=1053.414,307.982,-106.190,172.869,37.582,157.109
C01397=1053.421,308.230,-106.223,172.873,37.585,157.110
C01398=1053.427,308.478,-106.255,172.875,37.589,157.111
C01399=1053.434,308.724,-106.289,172.879,37.592,157.111
C01400=1053.440,308.973,-106.322,172.883,37.596,157.112
C01401=1053.447,309.220,-106.355,172.886,37.600,157.113
C01402=1053.454,309.469,-106.388,172.890,37.604,157.114
C01403=1053.460,309.716,-106.421,172.894,37.607,157.115
C01404=1053.467,309.964,-106.454,172.897,37.611,157.116
C01405=1053.473,310.212,-106.487,172.900,37.615,157.117
C01406=1053.481,310.459,-106.521,172.904,37.619,157.118
C01407=1053.487,310.707,-106.554,172.907,37.622,157.118
C01408=1053.495,310.954,-106.587,172.911,37.626,157.119
C01409=1053.501,311.202,-106.620,172.915,37.629,157.120
C01410=1053.508,311.449,-106.654,172.918,37.633,157.121
C01411=1053.515,311.697,-106.686,172.922,37.637,157.122
C01412=1053.521,311.945,-106.719,172.925,37.641,157.123
C01413=1053.528,312.192,-106.753,172.928,37.645,157.124
C01414=1053.535,312.441,-106.786,172.932,37.648,157.125
C01415=1053.542,312.688,-106.819,172.936,37.652,157.125
C01416=1053.548,312.936,-106.852,172.939,37.656,157.126
C01417=1053.555,313.183,-106.886,172.943,37.659,157.127
C01418=1053.562,313.430,-106.920,172.947,37.663,157.128
C01419=1053.568,313.678,-106.953,172.950,37.667,157.129
C01420=1053.575,313.926,-106.987,172.954,37.671,157.130
C01421=1053.581,314.173,-107.021,172.957,37.675,157.131
C01422=1053.588,314.422,-107.054,172.960,37.679,157.132
C01423=1053.594,314.669,-107.088,172.964,37.683,157.133
C01424=1053.601,314.917,-107.122,172.968,37.687,157.134
C01425=1053.607,315.164,-107.156,172.971,37.690,157.135
C01426=1053.614,315.412,-107.190,172.975,37.694,157.136
C01427=1053.619,315.659,-107.223,172.979,37.698,157.136
C01428=1053.627,315.907,-107.257,172.983,37.702,157.137
C01429=1053.633,316.154,-107.291,172.986,37.706,157.138
C01430=1053.640,316.402,-107.325,172.989,37.710,157.139
C01431=1053.646,316.649,-107.359,172.993,37.714,157.140
C01432=1053.653,316.897,-107.393,172.996,37.718,157.141
C01433=1053.659,317.145,-107.427,173.000,37.722,157.142
C01434=1053.666,317.392,-107.461,173.004,37.726,157.143
C01435=1053.672,317.641,-107.494,173.008,37.730,157.144
C01436=1053.679,317.888,-107.528,173.011,37.734,157.145
C01437=1053.686,318.165,-107.566,173.015,37.738,157.146
C01438=1053.693,318.443,-107.604,173.020,37.742,157.147
C01439=1053.702,318.720,-107.643,173.024,37.747,157.148
C01440=1053.708,318.996,-107.681,173.028,37.752,157.149
C01441=1053.715,319.244,-107.715,173.031,37.755,157.150
C01442=1053.722,319.492,-107.749,173.035,37.759,157.151
C01443=1053.728,319.739,-107.783,173.039,37.763,157.152
C01444=1053.735,319.987,-107.817,173.042,37.767,157.153
C01445=1053.742,320.235,-107.851,173.046,37.771,157.154
C01446=1053.747,320.482,-107.885,173.050,37.775,157.155
C01447=1053.755,320.730,-107.919,173.054,37.779,157.156
C01448=1053.761,320.978,-107.954,173.057,37.783,157.157
C01449=1053.769,321.225,-107.988,173.061,37.787,157.158
C01450=1053.774,321.472,-108.022,173.065,37.791,157.158
C01451=1053.782,321.720,-108.056,173.068,37.795,157.159
C01452=1053.788,321.968,-108.090,173.072,37.799,157.160
C01453=1053.795,322.215,-108.124,173.076,37.803,157.161
C01454=1053.802,322.463,-108.159,173.080,37.807,157.162
C01455=1053.808,322.710,-108.193,173.084,37.811,157.163
C01456=1053.815,322.958,-108.227,173.087,37.815,157.164
C01457=1053.822,323.206,-108.262,173.091,37.819,157.165
C01458=1053.829,323.453,-108.296,173.095,37.823,157.166
C01459=1053.836,323.701,-108.331,173.098,37.827,157.167
C01460=1053.841,323.948,-108.365,173.102,37.831,157.168
C01461=1053.849,324.195,-108.399,173.106,37.835,157.169
C01462=1053.855,324.443,-108.434,173.110,37.839,157.170
C01463=1053.863,324.690,-108.468,173.113,37.843,157.171
C01464=1053.869,324.938,-108.503,173.117,37.847,157.172
C01465=1053.876,325.186,-108.537,173.122,37.851,157.173
C01466=1053.883,325.433,-108.572,173.126,37.855,157.174
C01467=1053.890,325.681,-108.606,173.130,37.860,157.175
C01468=1053.897,325.928,-108.641,173.133,37.864,157.176
C01469=1053.904,326.176,-108.675,173.137,37.867,157.177
C01470=1053.911,326.424,-108.710,173.141,37.871,157.178
C01471=1053.918,326.671,-108.744,173.145,37.875,157.179
C01472=1053.925,326.919,-108.779,173.148,37.880,157.180
C01473=1053.931,327.166,-108.814,173.152,37.884,157.181
C01474=1053.939,327.414,-108.848,173.156,37.888,157.182
C01475=1053.945,327.661,-108.883,173.160,37.892,157.183
C01476=1053.952,327.909,-108.918,173.164,37.896,157.184
C01477=1053.959,328.156,-108.952,173.168,37.900,157.185
C01478=1053.966,328.403,-108.987,173.172,37.904,157.186
C01479=1053.972,328.651,-109.022,173.176,37.908,157.187
C01480=1053.980,328.898,-109.056,173.180,37.912,157.188
C01481=1053.987,329.146,-109.091,173.183,37.916,157.189
C01482=1053.993,329.394,-109.126,173.187,37.921,157.190
C01483=1054.001,329.641,-109.160,173.192,37.925,157.191
C01484=1054.007,329.888,-109.195,173.196,37.929,157.192
C01485=1054.014,330.136,-109.231,173.199,37.933,157.193
C01486=1054.021,330.383,-109.266,173.203,37.937,157.194
C01487=1054.028,330.630,-109.301,173.207,37.941,157.195
C01488=1054.034,330.878,-109.335,173.211,37.945,157.196
C01489=1054.041,331.126,-109.370,173.216,37.950,157.197
C01490=1054.048,331.373,-109.406,173.219,37.954,157.198
C01491=1054.055,331.620,-109.441,173.223,37.958,157.199
C01492=1054.061,331.868,-109.476,173.227,37.963,157.200
C01493=1054.067,332.091,-109.508,173.231,37.966,157.201
C01494=1054.074,332.313,-109.539,173.235,37.970,157.202
C01495=1054.080,332.536,-109.572,173.238,37.974,157.203
C01496=1054.086,332.759,-109.603,173.241,37.978,157.204
C01497=1054.093,332.982,-109.635,173.245,37.982,157.205
C01498=1054.098,333.204,-109.666,173.249,37.986,157.205
C01499=1054.104,333.427,-109.698,173.252,37.989,157.206
C01500=1054.111,333.649,-109.730,173.256,37.993,157.207
C01501=1054.117,333.897,-109.766,173.260,37.997,157.208
C01502=1054.124,334.144,-109.801,173.264,38.002,157.209
C01503=1054.131,334.393,-109.836,173.269,38.006,157.211
C01504=1054.138,334.639,-109.872,173.272,38.010,157.211
C01505=1054.145,334.887,-109.907,173.276,38.015,157.213
C01506=1054.152,335.134,-109.942,173.280,38.019,157.214
C01507=1054.158,335.381,-109.977,173.284,38.023,157.215
C01508=1054.166,335.629,-110.013,173.289,38.027,157.216
C01509=1054.173,335.876,-110.049,173.293,38.032,157.217
C01510=1054.180,336.124,-110.084,173.297,38.036,157.218
C01511=1054.186,336.371,-110.120,173.300,38.041,157.219
C01512=1054.193,336.619,-110.156,173.305,38.045,157.220
C01513=1054.200,336.866,-110.191,173.309,38.049,157.221
C01514=1054.207,337.113,-110.226,173.313,38.054,157.222
C01515=1054.213,337.360,-110.263,173.317,38.058,157.223
C01516=1054.221,337.609,-110.298,173.322,38.062,157.224
C01517=1054.228,337.855,-110.334,173.326,38.067,157.225
C01518=1054.234,338.103,-110.370,173.329,38.071,157.226
C01519=1054.241,338.350,-110.406,173.334,38.076,157.228
C01520=1054.248,338.598,-110.441,173.338,38.080,157.229
C01521=1054.255,338.845,-110.478,173.342,38.085,157.230
C01522=1054.261,339.092,-110.513,173.346,38.089,157.231
C01523=1054.269,339.340,-110.549,173.351,38.094,157.232
C01524=1054.275,339.587,-110.585,173.355,38.098,157.233
C01525=1054.282,339.834,-110.620,173.359,38.102,157.234
C01526=1054.290,340.081,-110.657,173.364,38.107,157.235
C01527=1054.296,340.329,-110.692,173.367,38.111,157.236
C01528=1054.303,340.576,-110.728,173.371,38.116,157.237
C01529=1054.311,340.823,-110.764,173.376,38.120,157.239
C01530=1054.317,341.071,-110.800,173.380,38.125,157.240
C01531=1054.324,341.318,-110.836,173.384,38.130,157.241
C01532=1054.331,341.566,-110.873,173.389,38.134,157.242
C01533=1054.338,341.812,-110.909,173.393,38.139,157.243
C01534=1054.345,342.060,-110.945,173.397,38.143,157.244
C01535=1054.351,342.307,-110.981,173.402,38.147,157.245
C01536=1054.359,342.555,-111.017,173.406,38.152,157.246
C01537=1054.366,342.802,-111.053,173.410,38.156,157.247
C01538=1054.373,343.049,-111.090,173.415,38.161,157.249
C01539=1054.379,343.296,-111.126,173.418,38.166,157.250
C01540=1054.387,343.544,-111.162,173.423,38.170,157.251
C01541=1054.393,343.791,-111.199,173.427,38.175,157.252
C01542=1054.400,344.038,-111.234,173.431,38.180,157.253
C01543=1054.407,344.285,-111.271,173.436,38.184,157.254
C01544=1054.414,344.532,-111.307,173.440,38.189,157.256
C01545=1054.421,344.780,-111.344,173.445,38.193,157.257
C01546=1054.428,345.027,-111.380,173.449,38.198,157.258
C01547=1054.435,345.274,-111.417,173.453,38.203,157.259
C01548=1054.446,345.670,-111.475,173.461,38.210,157.261
C01549=1054.458,346.086,-111.537,173.468,38.218,157.263
C01550=1054.465,346.353,-111.576,173.472,38.223,157.264
C01551=1054.473,346.621,-111.616,173.477,38.228,157.265
C01552=1054.481,346.889,-111.656,173.482,38.233,157.267
C01553=1054.488,347.136,-111.692,173.486,38.238,157.268
C01554=1054.494,347.384,-111.729,173.491,38.243,157.269
C01555=1054.502,347.631,-111.765,173.495,38.248,157.270
C01556=1054.509,347.877,-111.802,173.499,38.252,157.271
C01557=1054.516,348.125,-111.839,173.504,38.257,157.273
C01558=1054.523,348.373,-111.876,173.508,38.261,157.274
C01559=1054.530,348.619,-111.912,173.513,38.266,157.275
C01560=1054.537,348.867,-111.949,173.517,38.271,157.276
C01561=1054.544,349.115,-111.986,173.522,38.276,157.277
C01562=1054.551,349.361,-112.023,173.526,38.281,157.279
C01563=1054.558,349.608,-112.059,173.531,38.286,157.280
C01564=1054.565,349.856,-112.097,173.535,38.290,157.281
C01565=1054.572,350.103,-112.133,173.540,38.295,157.282
C01566=1054.579,350.350,-112.171,173.544,38.300,157.283
C01567=1054.587,350.597,-112.207,173.549,38.304,157.284
C01568=1054.594,350.844,-112.245,173.553,38.309,157.286
C01569=1054.600,351.091,-112.281,173.558,38.314,157.287
C01570=1054.608,351.339,-112.319,173.562,38.319,157.288
C01571=1054.615,351.586,-112.356,173.567,38.324,157.289
C01572=1054.621,351.833,-112.393,173.572,38.328,157.291
C01573=1054.628,352.080,-112.430,173.576,38.333,157.292
C01574=1054.636,352.327,-112.468,173.581,38.338,157.293
C01575=1054.643,352.574,-112.504,173.585,38.343,157.294
C01576=1054.650,352.821,-112.541,173.590,38.348,157.296
C01577=1054.657,353.068,-112.578,173.594,38.353,157.297
C01578=1054.664,353.315,-112.616,173.600,38.358,157.298
C01579=1054.672,353.562,-112.654,173.604,38.363,157.299
C01580=1054.679,353.810,-112.690,173.609,38.368,157.301
C01581=1054.685,354.056,-112.728,173.614,38.373,157.302
C01582=1054.692,354.304,-112.765,173.618,38.378,157.303
C01583=1054.700,354.551,-112.803,173.623,38.383,157.304
C01584=1054.707,354.798,-112.840,173.627,38.388,157.306
C01585=1054.714,355.045,-112.878,173.632,38.393,157.307
C01586=1054.721,355.292,-112.915,173.637,38.398,157.308
C01587=1054.729,355.539,-112.953,173.641,38.403,157.309
C01588=1054.736,355.786,-112.990,173.646,38.408,157.311
C01589=1054.742,356.033,-113.028,173.650,38.413,157.312
C01590=1054.749,356.280,-113.065,173.655,38.418,157.313
C01591=1054.756,356.527,-113.103,173.660,38.423,157.315
C01592=1054.764,356.775,-113.141,173.665,38.428,157.316
C01593=1054.771,357.022,-113.178,173.670,38.433,157.317
C01594=1054.778,357.269,-113.216,173.675,38.438,157.318
C01595=1054.786,357.515,-113.254,173.679,38.443,157.320
C01596=1054.793,357.762,-113.291,173.684,38.449,157.321
C01597=1054.800,358.010,-113.329,173.689,38.454,157.322
C01598=1054.807,358.257,-113.366,173.693,38.459,157.324
C01599=1054.815,358.503,-113.405,173.698,38.464,157.325
C01600=1054.821,358.751,-113.443,173.703,38.469,157.326
C01601=1054.829,358.998,-113.480,173.708,38.474,157.328
C01602=1054.836,359.244,-113.519,173.713,38.479,157.329
C01603=1054.843,359.491,-113.556,173.718,38.485,157.330
C01604=1054.850,359.739,-113.594,173.722,38.490,157.332
C01605=1054.859,360.012,-113.637,173.727,38.496,157.333
C01606=1054.867,360.284,-113.678,173.734,38.501,157.334
C01607=1054.874,360.557,-113.720,173.739,38.507,157.336
C01608=1054.883,360.830,-113.762,173.744,38.513,157.337
C01609=1054.890,361.077,-113.801,173.749,38.518,157.339
C01610=1054.897,361.324,-113.838,173.753,38.524,157.340
C01611=1054.904,361.571,-113.876,173.759,38.528,157.341
C01612=1054.911,361.818,-113.915,173.764,38.534,157.343
C01613=1054.918,362.065,-113.953,173.769,38.539,157.344
C01614=1054.927,362.312,-113.991,173.773,38.544,157.346
C01615=1054.934,362.559,-114.029,173.778,38.550,157.347
C01616=1054.941,362.806,-114.068,173.784,38.555,157.348
C01617=1054.948,363.053,-114.106,173.789,38.560,157.350
C01618=1054.956,363.299,-114.144,173.793,38.565,157.351
C01619=1054.963,363.547,-114.183,173.798,38.571,157.352
C01620=1054.970,363.794,-114.221,173.803,38.576,157.354
C01621=1054.977,364.041,-114.260,173.808,38.582,157.355
C01622=1054.985,364.287,-114.298,173.813,38.587,157.357
C01623=1054.992,364.534,-114.337,173.818,38.593,157.358
C01624=1054.998,364.781,-114.376,173.823,38.598,157.359
C01625=1055.007,365.028,-114.414,173.828,38.604,157.361
C01626=1055.013,365.275,-114.452,173.834,38.609,157.362
C01627=1055.021,365.522,-114.491,173.839,38.614,157.364
C01628=1055.027,365.769,-114.529,173.843,38.620,157.365
C01629=1055.036,366.016,-114.568,173.848,38.625,157.367
C01630=1055.043,366.262,-114.608,173.854,38.631,157.368
C01631=1055.049,366.509,-114.646,173.859,38.636,157.369
C01632=1055.057,366.756,-114.685,173.864,38.642,157.371
C01633=1055.064,367.003,-114.724,173.869,38.648,157.372
C01634=1055.072,367.250,-114.762,173.874,38.653,157.374
C01635=1055.079,367.496,-114.801,173.879,38.658,157.375
C01636=1055.087,367.744,-114.840,173.884,38.664,157.377
C01637=1055.094,367.990,-114.878,173.889,38.670,157.378
C01638=1055.102,368.237,-114.918,173.895,38.675,157.379
C01639=1055.109,368.484,-114.957,173.900,38.681,157.381
C01640=1055.116,368.731,-114.995,173.905,38.686,157.382
C01641=1055.124,368.978,-115.035,173.911,38.692,157.384
C01642=1055.131,369.224,-115.074,173.916,38.697,157.385
C01643=1055.139,369.472,-115.113,173.921,38.703,157.387
C01644=1055.146,369.717,-115.152,173.925,38.709,157.388
C01645=1055.153,369.964,-115.191,173.931,38.714,157.390
C01646=1055.161,370.212,-115.230,173.936,38.720,157.391
C01647=1055.168,370.458,-115.269,173.941,38.726,157.393
C01648=1055.176,370.705,-115.308,173.947,38.732,157.394
C01649=1055.183,370.951,-115.347,173.952,38.737,157.396
C01650=1055.191,371.199,-115.386,173.957,38.743,157.397
C01651=1055.198,371.445,-115.426,173.963,38.748,157.399
C01652=1055.206,371.692,-115.464,173.968,38.754,157.400
C01653=1055.214,371.939,-115.504,173.973,38.760,157.402
C01654=1055.221,372.185,-115.544,173.979,38.766,157.403
C01655=1055.229,372.433,-115.583,173.984,38.772,157.405
C01656=1055.236,372.679,-115.622,173.989,38.778,157.406
C01657=1055.244,372.926,-115.662,173.995,38.783,157.408
C01658=1055.251,373.172,-115.702,174.000,38.789,157.409
C01659=1055.258,373.420,-115.741,174.005,38.795,157.411
C01660=1055.265,373.666,-115.781,174.011,38.801,157.412
C01661=1055.274,373.957,-115.827,174.018,38.808,157.414
C01662=1055.283,374.249,-115.875,174.024,38.815,157.416
C01663=1055.292,374.540,-115.921,174.030,38.822,157.418
C01664=1055.301,374.832,-115.968,174.036,38.829,157.420
C01665=1055.309,375.079,-116.008,174.042,38.835,157.421
C01666=1055.316,375.326,-116.047,174.047,38.841,157.423
C01667=1055.323,375.572,-116.087,174.053,38.847,157.424
C01668=1055.331,375.819,-116.127,174.058,38.852,157.426
C01669=1055.339,376.066,-116.167,174.064,38.858,157.428
C01670=1055.346,376.311,-116.207,174.070,38.865,157.429
C01671=1055.354,376.558,-116.247,174.075,38.871,157.431
C01672=1055.362,376.805,-116.287,174.081,38.877,157.432
C01673=1055.369,377.051,-116.327,174.086,38.883,157.434
C01674=1055.377,377.298,-116.366,174.092,38.889,157.436
C01675=1055.384,377.545,-116.406,174.097,38.895,157.437
C01676=1055.392,377.791,-116.447,174.103,38.901,157.439
C01677=1055.400,378.038,-116.487,174.108,38.907,157.440
C01678=1055.407,378.285,-116.526,174.115,38.913,157.442
C01679=1055.415,378.531,-116.566,174.120,38.919,157.444
C01680=1055.423,378.778,-116.607,174.126,38.925,157.445
C01681=1055.431,379.025,-116.647,174.131,38.931,157.447
C01682=1055.438,379.272,-116.687,174.137,38.937,157.449
C01683=1055.446,379.518,-116.728,174.142,38.944,157.450
C01684=1055.454,379.765,-116.767,174.149,38.950,157.452
C01685=1055.462,380.011,-116.808,174.154,38.956,157.454
C01686=1055.469,380.257,-116.848,174.160,38.962,157.455
C01687=1055.477,380.504,-116.889,174.165,38.968,157.457
C01688=1055.484,380.751,-116.929,174.171,38.975,157.459
C01689=1055.492,380.997,-116.969,174.177,38.981,157.460
C01690=1055.500,381.244,-117.011,174.183,38.987,157.462
C01691=1055.507,381.491,-117.051,174.188,38.994,157.464
C01692=1055.515,381.737,-117.091,174.194,39.000,157.465
C01693=1055.523,381.983,-117.132,174.199,39.007,157.467
C01694=1055.531,382.230,-117.173,174.206,39.013,157.469
C01695=1055.538,382.477,-117.214,174.212,39.019,157.470
C01696=1055.546,382.723,-117.254,174.217,39.025,157.472
C01697=1055.554,382.969,-117.295,174.223,39.032,157.474
C01698=1055.561,383.216,-117.336,174.229,39.038,157.476
C01699=1055.569,383.462,-117.377,174.235,39.044,157.477
C01700=1055.577,383.709,-117.417,174.241,39.051,157.479
C01701=1055.584,383.955,-117.459,174.247,39.058,157.481
C01702=1055.592,384.202,-117.499,174.253,39.064,157.483
C01703=1055.600,384.448,-117.540,174.258,39.071,157.484
C01704=1055.608,384.694,-117.581,174.264,39.077,157.486
C01705=1055.616,384.941,-117.622,174.271,39.083,157.488
C01706=1055.623,385.187,-117.663,174.276,39.090,157.490
C01707=1055.631,385.434,-117.704,174.282,39.097,157.491
C01708=1055.639,385.680,-117.744,174.289,39.103,157.493
C01709=1055.646,385.926,-117.785,174.294,39.110,157.495
C01710=1055.655,386.173,-117.826,174.301,39.117,157.497
C01711=1055.663,386.419,-117.868,174.307,39.123,157.499
C01712=1055.671,386.666,-117.909,174.312,39.129,157.500
C01713=1055.679,386.912,-117.950,174.319,39.136,157.502
C01714=1055.686,387.159,-117.991,174.325,39.143,157.504
C01715=1055.695,387.405,-118.033,174.331,39.150,157.506
C01716=1055.702,387.652,-118.074,174.337,39.156,157.508
C01717=1055.713,387.975,-118.127,174.345,39.165,157.510
C01718=1055.723,388.298,-118.182,174.353,39.173,157.512
C01719=1055.734,388.621,-118.236,174.361,39.183,157.515
C01720=1055.744,388.944,-118.291,174.369,39.192,157.517
C01721=1055.752,389.191,-118.331,174.376,39.198,157.519
C01722=1055.761,389.437,-118.374,174.381,39.205,157.521
C01723=1055.769,389.684,-118.414,174.388,39.212,157.523
C01724=1055.777,389.930,-118.457,174.394,39.219,157.525
C01725=1055.784,390.176,-118.499,174.401,39.225,157.527
C01726=1055.792,390.422,-118.539,174.407,39.232,157.528
C01727=1055.801,390.669,-118.582,174.413,39.239,157.530
C01728=1055.808,390.915,-118.623,174.419,39.246,157.532
C01729=1055.816,391.161,-118.665,174.426,39.253,157.534
C01730=1055.825,391.407,-118.707,174.432,39.260,157.536
C01731=1055.832,391.654,-118.748,174.438,39.267,157.538
C01732=1055.840,391.901,-118.791,174.444,39.274,157.540
C01733=1055.849,392.146,-118.832,174.451,39.281,157.542
C01734=1055.857,392.393,-118.874,174.457,39.288,157.544
C01735=1055.864,392.639,-118.916,174.464,39.295,157.546
C01736=1055.873,392.886,-118.959,174.471,39.302,157.547
C01737=1055.881,393.131,-119.000,174.477,39.309,157.550
C01738=1055.889,393.378,-119.042,174.483,39.316,157.551
C01739=1055.897,393.624,-119.084,174.489,39.324,157.553
C01740=1055.905,393.870,-119.127,174.496,39.330,157.555
C01741=1055.913,394.116,-119.169,174.503,39.338,157.557
C01742=1055.921,394.363,-119.211,174.509,39.345,157.559
C01743=1055.929,394.609,-119.253,174.516,39.352,157.561
C01744=1055.937,394.855,-119.296,174.522,39.359,157.563
C01745=1055.946,395.101,-119.338,174.529,39.366,157.565
C01746=1055.954,395.347,-119.380,174.536,39.374,157.567
C01747=1055.962,395.594,-119.422,174.541,39.381,157.569
C01748=1055.970,395.840,-119.465,174.548,39.388,157.571
C01749=1055.978,396.086,-119.507,174.555,39.395,157.573
C01750=1055.986,396.332,-119.550,174.561,39.403,157.575
C01751=1055.995,396.579,-119.593,174.568,39.410,157.577
C01752=1056.002,396.824,-119.635,174.575,39.417,157.579
C01753=1056.011,397.071,-119.678,174.582,39.425,157.582
C01754=1056.019,397.317,-119.721,174.588,39.432,157.584
C01755=1056.027,397.563,-119.763,174.595,39.440,157.586
C01756=1056.035,397.809,-119.806,174.602,39.447,157.588
C01757=1056.044,398.055,-119.849,174.608,39.454,157.590
C01758=1056.052,398.301,-119.891,174.615,39.462,157.592
C01759=1056.060,398.547,-119.934,174.622,39.470,157.594
C01760=1056.068,398.794,-119.978,174.629,39.477,157.596
C01761=1056.076,399.039,-120.020,174.635,39.484,157.598
C01762=1056.084,399.286,-120.063,174.642,39.492,157.600
C01763=1056.093,399.532,-120.106,174.649,39.500,157.602
C01764=1056.101,399.778,-120.149,174.656,39.507,157.604
C01765=1056.110,400.024,-120.192,174.664,39.515,157.607
C01766=1056.118,400.270,-120.235,174.670,39.522,157.609
C01767=1056.127,400.516,-120.278,174.677,39.530,157.611
C01768=1056.135,400.762,-120.321,174.684,39.537,157.613
C01769=1056.143,401.008,-120.364,174.691,39.545,157.615
C01770=1056.152,401.255,-120.407,174.698,39.553,157.617
C01771=1056.160,401.501,-120.451,174.705,39.560,157.620
C01772=1056.169,401.747,-120.494,174.712,39.568,157.622
C01773=1056.180,402.088,-120.554,174.721,39.579,157.625
C01774=1056.192,402.429,-120.614,174.731,39.590,157.628
C01775=1056.203,402.770,-120.674,174.741,39.601,157.631
C01776=1056.215,403.111,-120.735,174.751,39.612,157.634
C01777=1056.223,403.357,-120.778,174.759,39.619,157.636
C01778=1056.232,403.604,-120.822,174.766,39.627,157.638
C01779=1056.241,403.849,-120.866,174.773,39.635,157.641
C01780=1056.249,404.095,-120.909,174.780,39.644,157.643
C01781=1056.257,404.341,-120.953,174.787,39.651,157.645
C01782=1056.266,404.587,-120.996,174.795,39.659,157.648
C01783=1056.274,404.833,-121.041,174.802,39.668,157.650
C01784=1056.283,405.079,-121.084,174.809,39.675,157.652
C01785=1056.291,405.325,-121.128,174.816,39.683,157.654
C01786=1056.300,405.571,-121.172,174.824,39.692,157.657
C01787=1056.308,405.817,-121.216,174.831,39.700,157.659
C01788=1056.317,406.063,-121.260,174.838,39.708,157.661
C01789=1056.325,406.309,-121.304,174.846,39.716,157.664
C01790=1056.333,406.555,-121.348,174.853,39.724,157.666
C01791=1056.342,406.801,-121.392,174.860,39.732,157.668
C01792=1056.350,407.047,-121.437,174.868,39.741,157.671
C01793=1056.359,407.292,-121.480,174.875,39.749,157.673
C01794=1056.368,407.538,-121.525,174.882,39.757,157.675
C01795=1056.376,407.784,-121.569,174.890,39.766,157.678
C01796=1056.385,408.030,-121.614,174.898,39.774,157.680
C01797=1056.393,408.276,-121.658,174.906,39.782,157.683
C01798=1056.402,408.521,-121.702,174.913,39.790,157.685
C01799=1056.411,408.768,-121.746,174.920,39.799,157.687
C01800=1056.419,409.014,-121.791,174.928,39.807,157.690
C01801=1056.428,409.260,-121.835,174.935,39.815,157.692
C01802=1056.437,409.506,-121.879,174.944,39.824,157.695
C01803=1056.445,409.751,-121.925,174.951,39.832,157.697
C01804=1056.455,409.998,-121.969,174.959,39.841,157.700
C01805=1056.463,410.243,-122.013,174.966,39.850,157.702
C01806=1056.472,410.489,-122.058,174.975,39.858,157.704
C01807=1056.481,410.735,-122.102,174.982,39.867,157.707
